	            //Year
	            #PieceID[23] := #is_ActualTime[1];
	            #PieceID[24] := #is_ActualTime[2];
	            #PieceID[25] := #is_ActualTime[3];
	            #PieceID[26] := #is_ActualTime[4];

	            //Month
	            #PieceID[27] := #is_ActualTime[6];
	            #PieceID[28] := #is_ActualTime[7];

	            //Day
	            #PieceID[29] := #is_ActualTime[9];
	            #PieceID[30] := #is_ActualTime[10];

	            //Constant
	            #PieceID[31] := '_';

	            //Time
	            #PieceID[32] := #is_ActualTime[12];
	            #PieceID[33] := #is_ActualTime[13];
	            #PieceID[34] := #is_ActualTime[14];
	            #PieceID[35] := #is_ActualTime[15];

	            //Constant
	            #PieceID[36] := '_';

	            //GIN
	            #ts_String := DELETE(IN := DINT_TO_STRING(#ii_GIN), L := 1, P := 1);

	            IF (#ii_GIN > 0) AND (#ii_GIN <= 9) THEN
	                #PieceID[37] := '0';
	                #PieceID[38] := '0';
	                #PieceID[39] := '0';
	                #PieceID[40] := #ts_String[1];
	            ELSIF (#ii_GIN >= 10) AND (#ii_GIN <= 99) THEN
	                #PieceID[37] := '0';
	                #PieceID[38] := '0';
	                #PieceID[39] := #ts_String[1];
	                #PieceID[40] := #ts_String[2];
	            ELSIF (#ii_GIN >= 100) AND (#ii_GIN <= 999) THEN
	                #PieceID[37] := '0';
	                #PieceID[38] := #ts_String[1];
	                #PieceID[39] := #ts_String[2];
	                #PieceID[40] := #ts_String[3];
	            ELSIF (#ii_GIN >= 1000) AND (#ii_GIN <= 9999) THEN
	                #PieceID[37] := #ts_String[1];
	                #PieceID[38] := #ts_String[2];
	                #PieceID[39] := #ts_String[3];
	                #PieceID[40] := #ts_String[4];
	            END_IF;

	            //Save data in DB GIN
	            "DB_GIN".GIN[#ii_GIN].DHL.PieceID := #PieceID;
	            "DB_GIN".GIN[#ii_GIN].DHL.VID := '000000000000000';

	            IF "DB_GIN".GIN[#ii_GIN].DHL.ObjectID = '' THEN
	                "DB_GIN".GIN[#ii_GIN].DHL.ObjectID := '0000000000';
	            END_IF;

	            //Generate a message to MFC
	            #FB_MFC_Sort_COY_ReceiveResult_Instance(is_VID := "DB_GIN".GIN[#ii_GIN].DHL.VID,
	                                                    is_PieceID := "DB_GIN".GIN[#ii_GIN].DHL.PieceID,
	                                                    is_Group := "DB_GIN".GIN[#ii_GIN].DHL.Xray.Group,
	                                                    is_Level := "DB_GIN".GIN[#ii_GIN].DHL.Xray.Level,
	                                                    is_Result := "DB_GIN".GIN[#ii_GIN].DHL.Xray.Result,
	                                                    ii_SourceNode := #ii_SourceNode,
	                                                    ii_DestinationNode := #ii_DestinationNode,
	                                                    iq_UDT_FifoHeader := #iq_UDT_FifoHeader,
	                                                    iqa_FifoData := #iqa_FifoData,
	                                                    iqi_MessageSequenceNumber := #iqi_MessageSequenceNumber);

	        END_IF;

	    END_IF;

	END_REGION

	REGION Parcel lost

	    //Check if parcel is lost in the tracking
	    //If there is, generate a message to MFC

	    IF #ii_GIN > 0 THEN

	        IF "DB_GIN".GIN[#ii_GIN].General.Lost THEN

	            //FORTNA internal exception results: L = Parcel lost
	            "DB_GIN".GIN[#ii_GIN].DHL.Xray.Result := 'L';

	            #FB_MFC_Sort_COY_ReceiveResult_Instance(is_VID := "DB_GIN".GIN[#ii_GIN].DHL.VID,
	                                                    is_PieceID := "DB_GIN".GIN[#ii_GIN].DHL.PieceID,
	                                                    is_Group := "DB_GIN".GIN[#ii_GIN].DHL.Xray.Group,
	                                                    is_Level := "DB_GIN".GIN[#ii_GIN].DHL.Xray.Level,
	                                                    is_Result := "DB_GIN".GIN[#ii_GIN].DHL.Xray.Result,
	                                                    ii_SourceNode := #ii_SourceNode,
	                                                    ii_DestinationNode := #ii_DestinationNode,
	                                                    iq_UDT_FifoHeader := #iq_UDT_FifoHeader,
	                                                    iqa_FifoData := #iqa_FifoData,
	                                                    iqi_MessageSequenceNumber := #iqi_MessageSequenceNumber);

	            //Save info in DB_GIN
	            "DB_GIN".GIN[#ii_GIN].DHL.MFCMessage.Sent.XrayResult := True;

	        END_IF;

	    END_IF;

	END_REGION

END_FUNCTION_BLOCK

FUNCTION_BLOCK "FB_MergeGINandObjectID"
{ S7_Optimized_Access := 'TRUE' }
VERSION : 0.1
// ATTRIBUTES
// AUTO_NUMBER = True
// BLOCK_NUMBER = 240
// END_ATTRIBUTES
   VAR_INPUT
      is_Configuration { ExternalAccessible := 'False'; ExternalVisible := 'False'; ExternalWritable := 'False'} : Struct   // Configuration
         SearchWindowStart { ExternalAccessible := 'False'; ExternalVisible := 'False'; ExternalWritable := 'False'} : Int;   // Start of the search window in conveyor tracking
         SearchWindowEnd { ExternalAccessible := 'False'; ExternalVisible := 'False'; ExternalWritable := 'False'} : Int;   // End of the search window in conveyor tracking
      END_STRUCT;
      iid_ReceivedObjectID { ExternalAccessible := 'False'; ExternalVisible := 'False'; ExternalWritable := 'False'} : DInt;   // Received ObjectID form sorter
      ia_ConveyorTracking { ExternalAccessible := 'False'; ExternalVisible := 'False'; ExternalWritable := 'False'} : Array[0..2501] of Int;   // ConveyorTracking
      ii_XrayLocation { ExternalAccessible := 'False'; ExternalVisible := 'False'; ExternalWritable := 'False'} : Int;   // X-ray location
      ii_SourceNode { ExternalAccessible := 'False'; ExternalVisible := 'False'; ExternalWritable := 'False'} : Int;   // ID Source Node
      ii_DestinationNode { ExternalAccessible := 'False'; ExternalVisible := 'False'; ExternalWritable := 'False'} : Int;   // ID Destination Node
   END_VAR

   VAR_IN_OUT
      iq_UDT_FifoHeader : "UDT_FifoHeader";   // FIFO header
      iqa_FifoData : Array[*] of "UDT_MessageV2";   // FIFO data buffer
      iqi_MessageSequenceNumber { ExternalAccessible := 'False'; ExternalVisible := 'False'; ExternalWritable := 'False'} : Int;   // Message number
   END_VAR

   VAR
      sid_ObjectID { ExternalAccessible := 'False'; ExternalVisible := 'False'; ExternalWritable := 'False'} : DInt;   // Saved Object ID
      sx_NewObjectID { ExternalAccessible := 'False'; ExternalVisible := 'False'; ExternalWritable := 'False'} : Bool;
      FB_MFC_Sort_COY_RegInfo_Instance { ExternalAccessible := 'False'; ExternalVisible := 'False'; ExternalWritable := 'False'; S7_SetPoint := 'False'} : "FB_MFC_Sort_COY_RegInfo";
   END_VAR

   VAR_TEMP
      ti_Loop : Int;
   END_VAR


BEGIN
	(*
	----------------------------------------------------------------------------------------
	|                                                                                      |
	|  Copyright  2023             FORTNA Europe BV                                        |
	|  All Rights Reserved         Netherlands                                             |
	|                                                                                      |
	----------------------------------------------------------------------------------------
	Version history:
	Date        | Version   | Author       | Remark
	----------------------------------------------------------------------------------------
	05/10/2023  | 1.0       | S. Nikodem   | Release TIA 17 | DHL Munich 2023
	13/03/2024  | 1.1       | S. Nieswiec  | Added to new Baseline
	*)

	REGION Save ObjectID

	    IF #iid_ReceivedObjectID <> #sid_ObjectID THEN

	        //New data
	        #sx_NewObjectID := True;

	        //Copy data to memory
	        #sid_ObjectID := #iid_ReceivedObjectID;

	    END_IF;

	END_REGION

	REGION Merge data

	    IF #sx_NewObjectID THEN

	        FOR #ti_Loop := #is_Configuration.SearchWindowStart TO #is_Configuration.SearchWindowEnd DO

	            IF #ia_ConveyorTracking[#ti_Loop] <> 0
	                AND ("DB_GIN".GIN[#ia_ConveyorTracking[#ti_Loop]].DHL.ObjectID = '')
	            THEN

	                //Combine data, save Object ID in DB GIN
	                "DB_GIN".GIN[#ia_ConveyorTracking[#ti_Loop]].DHL.ObjectID := DELETE(IN := DINT_TO_STRING(#sid_ObjectID), L := 1, P := 1);

	                //Data combined
	                #sx_NewObjectID := FALSE;

	                //Send a message to the MFC requesting information on the parcel
	                #FB_MFC_Sort_COY_RegInfo_Instance(is_ObjectID := "DB_GIN".GIN[#ia_ConveyorTracking[#ti_Loop]].DHL.ObjectID,
	                                                  ii_XrayLocation := #ii_XrayLocation,
	                                                  ii_SourceNode := #ii_SourceNode,
	                                                  ii_DestinationNode := #ii_DestinationNode,
	                                                  iq_UDT_FifoHeader := #iq_UDT_FifoHeader,
	                                                  iqa_FifoData := #iqa_FifoData,
	                                                  iqi_MessageSequenceNumber := #iqi_MessageSequenceNumber);

	                //Save information in DB GIN
	                "DB_GIN".GIN[#ia_ConveyorTracking[#ti_Loop]].DHL.MFCMessage.Sent.ParcelRegInfo := True;

	                //Exit loop
	                EXIT;

	            END_IF;

	        END_FOR;

	    END_IF;

	END_REGION
END_FUNCTION_BLOCK

FUNCTION_BLOCK "FB_SpecialHandlingArea"
TITLE = PLC0020 - DHL Munich
{ S7_Optimized_Access := 'TRUE' }
AUTHOR : 'R. Golonka'
VERSION : 0.1
// ATTRIBUTES
// AUTO_NUMBER = True
// BLOCK_NUMBER = 103
// END_ATTRIBUTES
//Block for special handling area
   VAR_INPUT
      i_UDT_ConveyorHandshakeUp { ExternalAccessible := 'False'; ExternalVisible := 'False'; ExternalWritable := 'False'} : "UDT_ConveyorHandshake";
      iudi_DelayTransferTime { ExternalAccessible := 'False'; ExternalVisible := 'False'; ExternalWritable := 'False'} : UDInt;   // Additional transfer time
      ix_KneeButton { ExternalAccessible := 'False'; ExternalVisible := 'False'; ExternalWritable := 'False'} : Bool;   // Input knee button conveyor 3
      ix_MannedButton { ExternalAccessible := 'False'; ExternalVisible := 'False'; ExternalWritable := 'False'} : Bool;   // Check in button to inform system about manned system
      ix_PEC_DownstreamEoS { ExternalAccessible := 'False'; ExternalVisible := 'False'; ExternalWritable := 'False'} : Bool;   // Downstream sensor end of section signal
      ix_PEC_EoS { ExternalAccessible := 'False'; ExternalVisible := 'False'; ExternalWritable := 'False'} : Bool;   // Sensor end of section signal
      ix_PEC_UpsteamEoS { ExternalAccessible := 'False'; ExternalVisible := 'False'; ExternalWritable := 'False'} : Bool;   // Upstream sensor end of section signal
      ix_LastStation { ExternalAccessible := 'False'; ExternalVisible := 'False'; ExternalWritable := 'False'} : Bool;   // Last station
   END_VAR

   VAR_OUTPUT
      q_UDT_HMIStatus { ExternalAccessible := 'False'; ExternalVisible := 'False'; ExternalWritable := 'False'} : "UDT_SHAStatus";   // SHA status
      qx_SygnalingLamp { ExternalAccessible := 'False'; ExternalVisible := 'False'; ExternalWritable := 'False'} : Bool;   // White lamp demmand
      qx_PushButtonLamp { ExternalAccessible := 'False'; ExternalVisible := 'False'; ExternalWritable := 'False'} : Bool;   // Push button lamp
      qx_ExternalDieback_1 { ExternalAccessible := 'False'; ExternalVisible := 'False'; ExternalWritable := 'False'} : Bool;   // External die back signal output
      qx_ExternalDieback_2 { ExternalAccessible := 'False'; ExternalVisible := 'False'; ExternalWritable := 'False'} : Bool;   // External die back signal output
      qx_ExternalDieback_3 { ExternalAccessible := 'False'; ExternalVisible := 'False'; ExternalWritable := 'False'} : Bool;   // External die back signal output
      qx_ExternalDiebackUp { ExternalAccessible := 'False'; ExternalVisible := 'False'; ExternalWritable := 'False'} : Bool;   // External die back signal output
   END_VAR

   VAR_IN_OUT
      iq_UDT_SHAInterfaceUp : "UDT_SHA_StationInterface";   // SHA interface
      iq_UDT_SHAInterface : "UDT_SHA_StationInterface";   // SHA interface
      iq_UDT_DownstreamConveyorHandshake : "UDT_ConveyorHandshake";   // Conveyor interface
      iq_UDT_ConveyorHandshake : "UDT_ConveyorHandshake";   // Conveyor interface
      iq_UDT_UpstreamConveyorHandshake : "UDT_ConveyorHandshake";   // Conveyor interface
   END_VAR

   VAR
      FB_TimerOnOffDelay_TransferInprogres { ExternalAccessible := 'False'; ExternalVisible := 'False'; ExternalWritable := 'False'; S7_SetPoint := 'False'} : "FB_TimerOnOffDelay";   // Additional timer time
      s_UDT_SHAInterface { ExternalAccessible := 'False'; ExternalVisible := 'False'; ExternalWritable := 'False'; S7_SetPoint := 'False'} : "UDT_SHA_StationInterface";   // Special handling area inteface
      s_UDT_HMIStatus { ExternalAccessible := 'False'; ExternalVisible := 'False'; ExternalWritable := 'False'; S7_SetPoint := 'False'} : "UDT_SHAStatus";   // SHA status
      R_TRIG_KneeButton {InstructionName := 'R_TRIG'; LibVersion := '1.0'; ExternalAccessible := 'False'; ExternalVisible := 'False'; ExternalWritable := 'False'; S7_SetPoint := 'False'} : R_TRIG;   // Rising edge knee button signal
      R_TRIG_MannedButton {InstructionName := 'R_TRIG'; LibVersion := '1.0'; ExternalAccessible := 'False'; ExternalVisible := 'False'; ExternalWritable := 'False'; S7_SetPoint := 'False'} : R_TRIG;   // Rising edge manned button signal
      R_TRIG_TIPUp {InstructionName := 'R_TRIG'; LibVersion := '1.0'; ExternalAccessible := 'False'; ExternalVisible := 'False'; ExternalWritable := 'False'; S7_SetPoint := 'False'} : R_TRIG;
      R_TRIG_TIPDown {InstructionName := 'R_TRIG'; LibVersion := '1.0'; ExternalAccessible := 'False'; ExternalVisible := 'False'; ExternalWritable := 'False'; S7_SetPoint := 'False'} : R_TRIG;
      R_TRIG_TIP {InstructionName := 'R_TRIG'; LibVersion := '1.0'; ExternalAccessible := 'False'; ExternalVisible := 'False'; ExternalWritable := 'False'; S7_SetPoint := 'False'} : R_TRIG;
      "#R_TRIG_RTSUp" {InstructionName := 'R_TRIG'; LibVersion := '1.0'; ExternalAccessible := 'False'; ExternalVisible := 'False'; ExternalWritable := 'False'; S7_SetPoint := 'False'} : R_TRIG;
      sx_SygnalingLamp { ExternalAccessible := 'False'; ExternalVisible := 'False'; ExternalWritable := 'False'} : Bool;   // White lamp demmand
      sx_PushButtonLamp { ExternalAccessible := 'False'; ExternalVisible := 'False'; ExternalWritable := 'False'} : Bool;   // Push button lamp
      sx_ExternalDieback_1 { ExternalAccessible := 'False'; ExternalVisible := 'False'; ExternalWritable := 'False'} : Bool;   // External dieback signal
      sx_ExternalDieback_2 { ExternalAccessible := 'False'; ExternalVisible := 'False'; ExternalWritable := 'False'} : Bool;   // External dieback signal
      sx_ExternalDieback_3 { ExternalAccessible := 'False'; ExternalVisible := 'False'; ExternalWritable := 'False'} : Bool;   // External dieback signal
      sx_ProductIsLocked { ExternalAccessible := 'False'; ExternalVisible := 'False'; ExternalWritable := 'False'} : Bool;   // Product is locked to the station
      sx_StationManned { ExternalAccessible := 'False'; ExternalVisible := 'False'; ExternalWritable := 'False'} : Bool;   // Station is occupied
      sx_DownstreamConveyorOccupied { ExternalAccessible := 'False'; ExternalVisible := 'False'; ExternalWritable := 'False'} : Bool;   // Downstream conveyor is occupied
      sx_MiddleConveyorOccupied { ExternalAccessible := 'False'; ExternalVisible := 'False'; ExternalWritable := 'False'} : Bool;   // Middle conveyor is occupied
      sx_UpstreamConveyorOccupied { ExternalAccessible := 'False'; ExternalVisible := 'False'; ExternalWritable := 'False'} : Bool;   // Upsteram conveyor is occupied
      si_NumberOfParcel { ExternalAccessible := 'False'; ExternalVisible := 'False'; ExternalWritable := 'False'} : Int;   // Number of parcel
      sx_ParcelTransfer { ExternalAccessible := 'False'; ExternalVisible := 'False'; ExternalWritable := 'False'} : Bool;   // Transfer in one section is in progress
      sx_ExternalDiebackUp { ExternalAccessible := 'False'; ExternalVisible := 'False'; ExternalWritable := 'False'} : Bool;   // Die back to previous station
   END_VAR


BEGIN
	(*
	----------------------------------------------------------------------------------------
	|                                                                                      |
	|  Copyright  2023             FORTNA Europe BV                                        |
	|  All Rights Reserved         Netherlands                                             |
	|                                                                                      |
	----------------------------------------------------------------------------------------
	Version history:
	Date        | Version   | Author       | Remark
	----------------------------------------------------------------------------------------
	06/10/2023  | 1.0       | R. Golonka   | Release TIA 17 | DHL Munich 2023
	13/03/2024  | 1.1       | S. Nieswiec  | Added to new baseline, block needs uptade after munich is finished
	*)

	REGION 1.0 - Inicialization
	    // Inicialization

	    #R_TRIG_KneeButton(CLK := #ix_KneeButton);
	    #R_TRIG_MannedButton(CLK := #ix_MannedButton);
	    #R_TRIG_TIPUp(CLK := #iq_UDT_UpstreamConveyorHandshake.TIP);
	    #R_TRIG_TIPDown(CLK := #iq_UDT_DownstreamConveyorHandshake.TIP);
	    #R_TRIG_TIP(CLK := #iq_UDT_ConveyorHandshake.TIP);
	    #"#R_TRIG_RTSUp"(CLK := #iq_UDT_ConveyorHandshake.RTS);

	END_REGION

	REGION 2.0 - Station manned

	    // Station in occupied (operator is working)
	    IF #R_TRIG_MannedButton.Q AND #iq_UDT_SHAInterfaceUp.Manned THEN

	        #sx_StationManned := NOT #sx_StationManned;
	        #sx_PushButtonLamp := NOT #sx_PushButtonLamp;

	    ELSIF (#iq_UDT_SHAInterfaceUp.Manned = false) THEN

	        #sx_StationManned := FALSE;
	        #sx_PushButtonLamp := FALSE;

	    ELSIF #ix_LastStation THEN

	        #sx_StationManned := #ix_LastStation;
	        #sx_PushButtonLamp := FALSE;

	    END_IF;

	END_REGION

	REGION 3.0 - Product locked and unlocked

	    // Product is locked in to the station
	    IF #R_TRIG_KneeButton.Q AND #sx_StationManned AND NOT #ix_PEC_DownstreamEoS THEN

	        #sx_ProductIsLocked := NOT #sx_ProductIsLocked;
	        #sx_SygnalingLamp := NOT #sx_SygnalingLamp;
	    ELSIF #R_TRIG_KneeButton.Q AND #sx_StationManned THEN
	        #sx_ProductIsLocked := false;
	        #sx_SygnalingLamp := false;
	    END_IF;

	END_REGION

	REGION 4.0 - Parcel in station

	    // Downstream station is occupied
	    #sx_DownstreamConveyorOccupied := NOT #ix_PEC_DownstreamEoS;
	    #sx_MiddleConveyorOccupied := NOT #ix_PEC_EoS;
	    #sx_UpstreamConveyorOccupied := NOT #ix_PEC_UpsteamEoS;

	    IF (#sx_DownstreamConveyorOccupied OR #sx_ProductIsLocked) THEN
	        #si_NumberOfParcel := 1;
	    END_IF;

	    IF (#sx_MiddleConveyorOccupied AND (#sx_DownstreamConveyorOccupied OR #sx_ProductIsLocked)) THEN
	        #si_NumberOfParcel := 2;
	    END_IF;

	    IF (#sx_UpstreamConveyorOccupied AND #sx_MiddleConveyorOccupied AND (#sx_DownstreamConveyorOccupied OR #sx_ProductIsLocked)) THEN
	        #si_NumberOfParcel := 3;
	    END_IF;

	    IF NOT #sx_UpstreamConveyorOccupied AND NOT #sx_MiddleConveyorOccupied AND NOT #sx_DownstreamConveyorOccupied THEN
	        #si_NumberOfParcel := 0;
	    END_IF;

	END_REGION

	REGION 5.0 - External dieback

	    IF #sx_StationManned
	        AND (#si_NumberOfParcel >= 3)
	        AND (#iq_UDT_SHAInterfaceUp.NumberOfParcel >= #si_NumberOfParcel)
	        AND #s_UDT_SHAInterface.Conveyor[2].Occupied
	        AND #s_UDT_SHAInterface.Conveyor[1].Occupied

	        OR #iq_UDT_SHAInterfaceUp.Conveyor[1].Locked
	        OR #sx_ProductIsLocked
	    THEN
	        #sx_ExternalDieback_1 := TRUE;
	    ELSE
	        #sx_ExternalDieback_1 := FALSE;
	    END_IF;

	    IF #sx_StationManned
	        AND (#si_NumberOfParcel >= 2)
	        AND (#iq_UDT_SHAInterfaceUp.NumberOfParcel >= #si_NumberOfParcel)
	        AND #s_UDT_SHAInterface.Conveyor[1].Occupied

	        OR #iq_UDT_SHAInterfaceUp.Conveyor[1].Locked
	        OR #sx_ProductIsLocked
	    THEN
	        #sx_ExternalDieback_2 := TRUE;
	    ELSE
	        #sx_ExternalDieback_2 := FALSE;
	    END_IF;

	    IF #sx_StationManned
	        AND (#si_NumberOfParcel >= 1)
	        AND (#iq_UDT_SHAInterfaceUp.NumberOfParcel >= #si_NumberOfParcel)
	        AND NOT #ix_PEC_DownstreamEoS
	        AND #iq_UDT_SHAInterfaceUp.Conveyor[1].Occupied
	        //AND #iq_UDT_SHAInterfaceUp.NumberOfParcel <> 0
	        OR #iq_UDT_SHAInterfaceUp.Conveyor[1].Locked
	        OR #sx_ProductIsLocked
	    THEN
	        #sx_ExternalDieback_3 := TRUE;
	    ELSIF #sx_StationManned AND (NOT #ix_PEC_DownstreamEoS AND #ix_LastStation) THEN
	        #sx_ExternalDieback_3 := TRUE;
	    ELSE
	        #sx_ExternalDieback_3 := FALSE;
	    END_IF;

	END_REGION

	REGION 8.0 - Reset RTR

	    // Set RTR to run conveyor

	    IF NOT #sx_DownstreamConveyorOccupied AND #ix_KneeButton AND #sx_StationManned THEN
	        #iq_UDT_DownstreamConveyorHandshake.RTR := true;
	    END_IF;

	    IF NOT #sx_MiddleConveyorOccupied AND #ix_KneeButton AND #sx_StationManned THEN
	        #iq_UDT_ConveyorHandshake.RTR := true;
	    END_IF;

	    IF NOT #sx_UpstreamConveyorOccupied AND #ix_KneeButton AND #sx_StationManned THEN
	        #iq_UDT_UpstreamConveyorHandshake.RTR := true;
	    END_IF;

	END_REGION

	REGION 7.0 - Hold for previous station when station is in transfer

	    #sx_ParcelTransfer := (#R_TRIG_KneeButton.Q)
	    OR (#R_TRIG_TIPDown.Q)
	    OR (#R_TRIG_TIP.Q)
	    OR (#R_TRIG_TIPUp.Q);

	    #FB_TimerOnOffDelay_TransferInprogres(iudi_OffDelayTime := #iudi_DelayTransferTime,
	                                          ix_SignalToDelay := #sx_ParcelTransfer,
	                                          ix_Enable := TRUE,
	                                          qx_DelayedSignal => #sx_ExternalDiebackUp);

	END_REGION

	REGION 8.0 - Update Interface

	    #s_UDT_SHAInterface.Manned := #sx_StationManned;
	    #s_UDT_SHAInterface.NumberOfParcel := #si_NumberOfParcel;
	    #s_UDT_SHAInterface.TransferInProgres := #sx_ParcelTransfer;
	    #s_UDT_SHAInterface.Conveyor[1].Empty := NOT #sx_DownstreamConveyorOccupied;
	    #s_UDT_SHAInterface.Conveyor[1].Locked := #sx_ProductIsLocked;
	    #s_UDT_SHAInterface.Conveyor[1].Occupied := #sx_DownstreamConveyorOccupied;
	    #s_UDT_SHAInterface.Conveyor[2].Empty := NOT #sx_MiddleConveyorOccupied;
	    #s_UDT_SHAInterface.Conveyor[2].Locked := FALSE;
	    #s_UDT_SHAInterface.Conveyor[2].Occupied := #sx_MiddleConveyorOccupied;
	    #s_UDT_SHAInterface.Conveyor[3].Empty := NOT #sx_UpstreamConveyorOccupied;
	    #s_UDT_SHAInterface.Conveyor[3].Locked := FALSE;
	    #s_UDT_SHAInterface.Conveyor[3].Occupied := #sx_UpstreamConveyorOccupied;

	END_REGION

	REGION 9.0 - Status

	    // Status half full
	    #s_UDT_HMIStatus.Specific.HalfFull := #sx_StationManned AND (#s_UDT_SHAInterface.NumberOfParcel >= 3);
	    // Status full
	    #s_UDT_HMIStatus.Specific.Full := #sx_StationManned AND (#iq_UDT_SHAInterfaceUp.NumberOfParcel >= 3) AND (#s_UDT_SHAInterface.NumberOfParcel >= 3) AND #i_UDT_ConveyorHandshakeUp.RTS;

	    // HMI status initialization
	    #s_UDT_HMIStatus.Status := 0;

	    // Copy HMI status to output
	    #q_UDT_HMIStatus := #s_UDT_HMIStatus;

	END_REGION

	REGION 10.0 - Output

	    // Output write
	    #qx_ExternalDieback_1 := #sx_ExternalDieback_1;
	    #qx_ExternalDieback_2 := #sx_ExternalDieback_2;
	    #qx_ExternalDieback_3 := #sx_ExternalDieback_3;
	    #qx_ExternalDiebackUp := #sx_ExternalDiebackUp AND #i_UDT_ConveyorHandshakeUp.RTS;
	    #qx_SygnalingLamp := #sx_SygnalingLamp;
	    #qx_PushButtonLamp := #sx_PushButtonLamp;
	    #iq_UDT_SHAInterface := #s_UDT_SHAInterface;

	END_REGION
END_FUNCTION_BLOCK

FUNCTION_BLOCK "FB_SNCY_InfeedControlPanel"
{ S7_Optimized_Access := 'TRUE' }
VERSION : 0.1
// ATTRIBUTES
// AUTO_NUMBER = True
// BLOCK_NUMBER = 102
// END_ATTRIBUTES
   VAR_INPUT
      ix_InfeedButton { ExternalAccessible := 'False'; ExternalVisible := 'False'; ExternalWritable := 'False'} : Bool;   // Signal from infeed push button
      ix_OutfeedButton { ExternalAccessible := 'False'; ExternalVisible := 'False'; ExternalWritable := 'False'} : Bool;   // Signal from outfeed push button
      i_UDT_ExitConveyorStatus { ExternalAccessible := 'False'; ExternalVisible := 'False'; ExternalWritable := 'False'} : "UDT_CommonStatus";   // Common status from outfeed exit conveyor
      ix_InfeedModeActive { ExternalAccessible := 'False'; ExternalVisible := 'False'; ExternalWritable := 'False'} : Bool;   // True - when infeed mode is active
      ix_OutfeedModeActive { ExternalAccessible := 'False'; ExternalVisible := 'False'; ExternalWritable := 'False'} : Bool;   // True - when outfeed mode is active
   END_VAR

   VAR_OUTPUT
      qx_InfeedLamp { ExternalAccessible := 'False'; ExternalVisible := 'False'; ExternalWritable := 'False'} : Bool;   // Lamp for Infeed status
      qx_OutfeedLamp { ExternalAccessible := 'False'; ExternalVisible := 'False'; ExternalWritable := 'False'} : Bool;   // Lamp for Outfeed status
      qx_ConveyorHold { ExternalAccessible := 'False'; ExternalVisible := 'False'; ExternalWritable := 'False'} : Bool;   // Conveyor hold command for associated conveyor
   END_VAR

   VAR
      R_TRIG_ToogleInfeedButton {InstructionName := 'R_TRIG'; LibVersion := '1.0'; ExternalAccessible := 'False'; ExternalVisible := 'False'; ExternalWritable := 'False'; S7_SetPoint := 'False'} : R_TRIG;   // Rising edge trigger infeed button
      R_TRIG_ToogleOutfeedButton {InstructionName := 'R_TRIG'; LibVersion := '1.0'; ExternalAccessible := 'False'; ExternalVisible := 'False'; ExternalWritable := 'False'; S7_SetPoint := 'False'} : R_TRIG;   // Rising edge trigger outfeed button
      R_TRIG_Modeline {InstructionName := 'R_TRIG'; LibVersion := '1.0'; ExternalAccessible := 'False'; ExternalVisible := 'False'; ExternalWritable := 'False'; S7_SetPoint := 'False'} : R_TRIG;   // Rising edge trigger mode line
      sx_SectionHold { ExternalAccessible := 'False'; ExternalVisible := 'False'; ExternalWritable := 'False'} : Bool;
   END_VAR


BEGIN
	(*
	----------------------------------------------------------------------------------------
	|                                                                                      |
	|  Copyright  2023             Fortna Europe BV                                        |
	|  All Rights Reserved         Netherlands                                             |
	|                                                                                      |
	|                                                                                      |
	----------------------------------------------------------------------------------------

	Version history:
	Date        | Version   | Author       | Remark
	----------------------------------------------------------------------------------------
	18/10/2023  | 1.0       | S. Nikodem   | Release TIA 17 | DHL Munich 2023
	13/03/2024  | 1.1       | S. Nieswiec  | Added to new baseline, block needs uptade after munich is finished
	*)

	REGION Buttons

	    //Infeed
	    IF #ix_InfeedModeActive THEN

	        #R_TRIG_ToogleInfeedButton(CLK := (#ix_InfeedButton));

	        IF #R_TRIG_ToogleInfeedButton.Q THEN

	            #sx_SectionHold := NOT #sx_SectionHold;

	        END_IF;

	    END_IF;

	    //Outfeed
	    IF #ix_OutfeedModeActive THEN

	        #R_TRIG_ToogleOutfeedButton(CLK := (#ix_OutfeedButton));

	        IF #R_TRIG_ToogleOutfeedButton.Q THEN

	            #sx_SectionHold := NOT #sx_SectionHold;

	        END_IF;

	    END_IF;

	END_REGION

	REGION Lamps

	    //Infeed
	    IF #ix_InfeedModeActive THEN

	        IF #sx_SectionHold THEN
	            #qx_InfeedLamp := "DB_Memory".Clock_1Hz;
	        ELSE
	            #qx_InfeedLamp := TRUE;
	        END_IF;

	    ELSE
	        #qx_InfeedLamp := False;
	    END_IF;

	    //Outfeed
	    IF #ix_OutfeedModeActive THEN

	        IF #sx_SectionHold THEN
	            #qx_OutfeedLamp := "DB_Memory".Clock_1Hz;
	        ELSE
	            #qx_OutfeedLamp := TRUE;
	        END_IF;

	    ELSE
	        #qx_OutfeedLamp := False;
	    END_IF;

	END_REGION

	REGION Conveyor hold command

	    #qx_ConveyorHold := #sx_SectionHold;

	END_REGION

	REGION Reset

	    //Reset when mode line is changed
	    #R_TRIG_Modeline(CLK := #ix_InfeedModeActive OR #ix_OutfeedModeActive);

	    IF #R_TRIG_Modeline.Q THEN
	        // Statement section IF
	        ;
	    END_IF;


	END_REGION



END_FUNCTION_BLOCK

FUNCTION_BLOCK "FB_SNCY_ArmDiverter"
{ S7_Optimized_Access := 'TRUE' }
VERSION : 0.1
// ATTRIBUTES
// AUTO_NUMBER = True
// BLOCK_NUMBER = 241
// END_ATTRIBUTES
   VAR_INPUT
      i_UDT_DiverterArmConfig { ExternalAccessible := 'False'; ExternalVisible := 'False'; ExternalWritable := 'False'} : "UDT_ArmDiverterConfiguration";   // Diverter arm configuration
      ix_SafetyOk { ExternalAccessible := 'False'; ExternalVisible := 'False'; ExternalWritable := 'False'} : Bool;   // TRUE when safety is ok
      ix_24vOk { ExternalAccessible := 'False'; ExternalVisible := 'False'; ExternalWritable := 'False'} : Bool;   // TRUE when 24VDC is healthy
      ix_400vOk { ExternalAccessible := 'False'; ExternalVisible := 'False'; ExternalWritable := 'False'} : Bool;   // TRUE when 400VAC is healthy
      ix_HardwareOk { ExternalAccessible := 'False'; ExternalVisible := 'False'; ExternalWritable := 'False'} : Bool;   // TRUE when  hardware is Ok
      ix_PRX_Home { ExternalAccessible := 'False'; ExternalVisible := 'False'; ExternalWritable := 'False'} : Bool;   // Proxy sensor home position
      ix_PRX_Divert { ExternalAccessible := 'False'; ExternalVisible := 'False'; ExternalWritable := 'False'} : Bool;   // Proxy sensor divert position
      ix_LS_Home { ExternalAccessible := 'False'; ExternalVisible := 'False'; ExternalWritable := 'False'} : Bool;   // Limit switch home position
      ix_LS_Divert { ExternalAccessible := 'False'; ExternalVisible := 'False'; ExternalWritable := 'False'} : Bool;   // Limit switch divert position
      ix_PRX_BRK_Home { ExternalAccessible := 'False'; ExternalVisible := 'False'; ExternalWritable := 'False'} : Bool;   // Brake sensor divert
      ix_PRX_BRK_Divert { ExternalAccessible := 'False'; ExternalVisible := 'False'; ExternalWritable := 'False'} : Bool;   // Brake sensor home
      ix_PEC_Exit { ExternalAccessible := 'False'; ExternalVisible := 'False'; ExternalWritable := 'False'} : Bool;   // TRUE when PEC Exit is not blocked
      ii_SourceNode { ExternalAccessible := 'False'; ExternalVisible := 'False'; ExternalWritable := 'False'} : Int := 0;   // Source Node
      ii_DestinationNode { ExternalAccessible := 'False'; ExternalVisible := 'False'; ExternalWritable := 'False'} : Int := 0;   // Destination Node
   END_VAR

   VAR_OUTPUT
      q_UDT_HMIStatus { ExternalAccessible := 'False'; ExternalVisible := 'False'; ExternalWritable := 'False'} : "UDT_ArmDiverterStatus";   // HMI status structure
      q_UDT_Status { ExternalAccessible := 'False'; ExternalVisible := 'False'; ExternalWritable := 'False'} : "UDT_CommonStatus";   // Common status structure
      qx_VerticalConveyorHold { ExternalAccessible := 'False'; ExternalVisible := 'False'; ExternalWritable := 'False'} : Bool;   // Command stop Vertical conveyor
      qx_AssociatedConveyorHold { ExternalAccessible := 'False'; ExternalVisible := 'False'; ExternalWritable := 'False'} : Bool;   // Command stop Associated conveyor
   END_VAR

   VAR_IN_OUT
      iq_UDT_EquipmentControl : "UDT_EquipmentControl";   // Equipment control structure
      iq_UDT_AssociatedConveyorInterface : "UDT_ConveyorInterface";   // Sorter main conveyor interface
      iq_UDT_VerticalConveyorInterface : "UDT_ConveyorInterface";   // Arm vertical conveyor interafce
      iq_UDT_ArmConveyorInterface : "UDT_ConveyorInterface";   // Arm conveyor interface
      iq_UDT_AssociatedConveyorHandshake : "UDT_ConveyorHandshake";   // Handshake structure
      iq_UDT_ExitConveyorHandshake : "UDT_ConveyorHandshake";   // Exit conveyor handshake structure
      iqa_AssociatedTrackingData : Array[*] of Int;   // Tracking data from sorter conveyor
      iqa_OutfeedsStatus : Array[*] of "UDT_OutfeedStatus";   // Structure with outfeeds status
      iq_UDT_ArmDiverterCommand : "UDT_ArmDiverterCommand";   // Arm Diverter command structure
      iq_UDT_FifoHeader_MFCMessage : "UDT_FifoHeader";   // MFC Message FIFO header
      iqs_FifoData_MFCMessage : Array[*] of "UDT_MessageV2";   // MFC Message FIFO data buffer
      iqdi_MessageSequenceNumber { ExternalAccessible := 'False'; ExternalVisible := 'False'; ExternalWritable := 'False'} : Int;   // MFC Message Message number
   END_VAR

   VAR
      FB_MFC_Sort_SortResult_HigherPriorityAvailable { ExternalAccessible := 'False'; ExternalVisible := 'False'; ExternalWritable := 'False'; S7_SetPoint := 'False'} : "FB_MFC_Sort_SortResult";   // Function to MFC message generation
      FB_MFC_Sort_SortResult { ExternalAccessible := 'False'; ExternalVisible := 'False'; ExternalWritable := 'False'; S7_SetPoint := 'False'} : "FB_MFC_Sort_SortResult";   // Function to MFC message generation
      FB_MFC_Sort_SortResult_Instance { ExternalAccessible := 'False'; ExternalVisible := 'False'; ExternalWritable := 'False'; S7_SetPoint := 'False'} : "FB_MFC_Sort_SortResult";   // Function to MFC message generation
      s_FB_PRX_HomeFiltered { ExternalAccessible := 'False'; ExternalVisible := 'False'; ExternalWritable := 'False'; S7_SetPoint := 'False'} : "FB_TimerOnOffDelay";   // Filtering proxy sensor home position signal
      s_FB_PRX_DivertFiltered { ExternalAccessible := 'False'; ExternalVisible := 'False'; ExternalWritable := 'False'; S7_SetPoint := 'False'} : "FB_TimerOnOffDelay";   // Filtering proxy sensor divert position signal
      s_FB_LS_HomeFiltered { ExternalAccessible := 'False'; ExternalVisible := 'False'; ExternalWritable := 'False'; S7_SetPoint := 'False'} : "FB_TimerOnOffDelay";   // Filtering limit switch home position signal
      s_FB_LS_DivertFiltered { ExternalAccessible := 'False'; ExternalVisible := 'False'; ExternalWritable := 'False'; S7_SetPoint := 'False'} : "FB_TimerOnOffDelay";   // Filtering limit switch divert position signal
      s_FB_BRK_PRX_HomeFiltered { ExternalAccessible := 'False'; ExternalVisible := 'False'; ExternalWritable := 'False'; S7_SetPoint := 'False'} : "FB_TimerOnOffDelay";   // Filtering proxy sensor home position signal
      s_FB_BRK_PRX_DivertFiltered { ExternalAccessible := 'False'; ExternalVisible := 'False'; ExternalWritable := 'False'; S7_SetPoint := 'False'} : "FB_TimerOnOffDelay";   // Filtering proxy sensor divert position signal
      s_FB_TimeoutError { ExternalAccessible := 'False'; ExternalVisible := 'False'; ExternalWritable := 'False'; S7_SetPoint := 'False'} : "FB_TimerOnOffDelay";   // Movement timeout error
      s_FB_Jog_Enable { ExternalAccessible := 'False'; ExternalVisible := 'False'; ExternalWritable := 'False'; S7_SetPoint := 'False'} : "FB_TimerOnOffDelay";   // Filtering lower jam photo eye signal
      s_FB_DivertTime { ExternalAccessible := 'False'; ExternalVisible := 'False'; ExternalWritable := 'False'; S7_SetPoint := 'False'} : "FB_TimerOnOffDelay";   // Divert time
      s_FB_InhibitTimeFilter { ExternalAccessible := 'False'; ExternalVisible := 'False'; ExternalWritable := 'False'; S7_SetPoint := 'False'} : "FB_TimerOnOffDelay";   // Filtering inhibit stop
      s_UDT_CommonStatus { ExternalAccessible := 'False'; ExternalVisible := 'False'; ExternalWritable := 'False'; S7_SetPoint := 'False'} : "UDT_CommonStatus";   // Common status structure
      s_UDT_CommonStatusOld { ExternalAccessible := 'False'; ExternalVisible := 'False'; ExternalWritable := 'False'; S7_SetPoint := 'False'} : "UDT_CommonStatus";   // Auxiliary status structure
      s_UDT_HMIStatus { ExternalAccessible := 'False'; ExternalVisible := 'False'; ExternalWritable := 'False'; S7_SetPoint := 'False'} : "UDT_ArmDiverterStatus";   // HMI status structure
      R_TRIG_ManualJogHome {InstructionName := 'R_TRIG'; LibVersion := '1.0'; ExternalAccessible := 'False'; ExternalVisible := 'False'; ExternalWritable := 'False'; S7_SetPoint := 'False'} : R_TRIG;   // Rising edge trigger manual jog mode command
      R_TRIG_ManualJogDivert {InstructionName := 'R_TRIG'; LibVersion := '1.0'; ExternalAccessible := 'False'; ExternalVisible := 'False'; ExternalWritable := 'False'; S7_SetPoint := 'False'} : R_TRIG;   // Rising edge trigger manual jog mode command
      R_TRIG_PRX_Home {InstructionName := 'R_TRIG'; LibVersion := '1.0'; ExternalAccessible := 'False'; ExternalVisible := 'False'; ExternalWritable := 'False'; S7_SetPoint := 'False'} : R_TRIG;   // Rising edge trigger
      R_TRIG_PRX_Divert {InstructionName := 'R_TRIG'; LibVersion := '1.0'; ExternalAccessible := 'False'; ExternalVisible := 'False'; ExternalWritable := 'False'; S7_SetPoint := 'False'} : R_TRIG;   // Rising edge trigger
      R_TRIG_LS_Home {InstructionName := 'R_TRIG'; LibVersion := '1.0'; ExternalAccessible := 'False'; ExternalVisible := 'False'; ExternalWritable := 'False'; S7_SetPoint := 'False'} : R_TRIG;   // Rising edge trigger
      R_TRIG_LS_Divert {InstructionName := 'R_TRIG'; LibVersion := '1.0'; ExternalAccessible := 'False'; ExternalVisible := 'False'; ExternalWritable := 'False'; S7_SetPoint := 'False'} : R_TRIG;   // Rising edge trigger
      F_TRIG_PRX_Home {InstructionName := 'F_TRIG'; LibVersion := '1.0'; ExternalAccessible := 'False'; ExternalVisible := 'False'; ExternalWritable := 'False'; S7_SetPoint := 'False'} : F_TRIG;   // Falling edge trigger
      F_TRIG_PRX_Divert {InstructionName := 'F_TRIG'; LibVersion := '1.0'; ExternalAccessible := 'False'; ExternalVisible := 'False'; ExternalWritable := 'False'; S7_SetPoint := 'False'} : F_TRIG;   // Falling edge trigger
      F_TRIG_LS_Home {InstructionName := 'F_TRIG'; LibVersion := '1.0'; ExternalAccessible := 'False'; ExternalVisible := 'False'; ExternalWritable := 'False'; S7_SetPoint := 'False'} : F_TRIG;   // Falling edge trigger
      F_TRIG_LS_Divert {InstructionName := 'F_TRIG'; LibVersion := '1.0'; ExternalAccessible := 'False'; ExternalVisible := 'False'; ExternalWritable := 'False'; S7_SetPoint := 'False'} : F_TRIG;   // Falling edge trigger
      F_TRIG_BRK_PRX_Home {InstructionName := 'F_TRIG'; LibVersion := '1.0'; ExternalAccessible := 'False'; ExternalVisible := 'False'; ExternalWritable := 'False'; S7_SetPoint := 'False'} : F_TRIG;   // Falling edge trigger
      R_TRIG_BRK_PRX_Home {InstructionName := 'R_TRIG'; LibVersion := '1.0'; ExternalAccessible := 'False'; ExternalVisible := 'False'; ExternalWritable := 'False'; S7_SetPoint := 'False'} : R_TRIG;   // Rising edge trigger
      F_TRIG_BRK_PRX_Divert {InstructionName := 'F_TRIG'; LibVersion := '1.0'; ExternalAccessible := 'False'; ExternalVisible := 'False'; ExternalWritable := 'False'; S7_SetPoint := 'False'} : F_TRIG;   // Falling edge trigger
      R_TRIG_BRK_PRX_Divert {InstructionName := 'R_TRIG'; LibVersion := '1.0'; ExternalAccessible := 'False'; ExternalVisible := 'False'; ExternalWritable := 'False'; S7_SetPoint := 'False'} : R_TRIG;   // Rising edge trigger
      R_TRIG_ExitSensor {InstructionName := 'R_TRIG'; LibVersion := '1.0'; ExternalAccessible := 'False'; ExternalVisible := 'False'; ExternalWritable := 'False'; S7_SetPoint := 'False'} : R_TRIG;   // Rising edge trigger of exit sensor
      F_TRIG_ArmConveyorLowSpeed {InstructionName := 'F_TRIG'; LibVersion := '1.0'; ExternalAccessible := 'False'; ExternalVisible := 'False'; ExternalWritable := 'False'; S7_SetPoint := 'False'} : F_TRIG;   // Falling edge trigger
      R_TRIG_ParcelLocation {InstructionName := 'R_TRIG'; LibVersion := '1.0'; ExternalAccessible := 'False'; ExternalVisible := 'False'; ExternalWritable := 'False'; S7_SetPoint := 'False'} : R_TRIG;   // Rising edge trigger
      ss_Counter { ExternalAccessible := 'False'; ExternalVisible := 'False'; ExternalWritable := 'False'} : Struct   // Counters for statistics
         ParcelDetected { ExternalAccessible := 'False'; ExternalVisible := 'False'; ExternalWritable := 'False'} : UDInt;   // New package was detected
         ParcelInWindow { ExternalAccessible := 'False'; ExternalVisible := 'False'; ExternalWritable := 'False'} : UDInt;   // Another parcel is within the range of arm movement. The parcel cannot be sorted.
         SortParcelCommand { ExternalAccessible := 'False'; ExternalVisible := 'False'; ExternalWritable := 'False'} : UDInt;
         SortResultMessage { ExternalAccessible := 'False'; ExternalVisible := 'False'; ExternalWritable := 'False'} : UDInt;
         LoopExit { ExternalAccessible := 'False'; ExternalVisible := 'False'; ExternalWritable := 'False'} : UDInt;
      END_STRUCT;
      ss_SortStrategy { ExternalAccessible := 'False'; ExternalVisible := 'False'; ExternalWritable := 'False'} : Struct   // Sort Strategy
         HigherPriorityAvailable { ExternalAccessible := 'False'; ExternalVisible := 'False'; ExternalWritable := 'False'} : Bool;
         ObjectID { ExternalAccessible := 'False'; ExternalVisible := 'False'; ExternalWritable := 'False'} : String[10];
      END_STRUCT;
      ss_SortedObjectID { ExternalAccessible := 'False'; ExternalVisible := 'False'; ExternalWritable := 'False'} : String[10];   // Stored value of the last Object ID
      si_GINSort { ExternalAccessible := 'False'; ExternalVisible := 'False'; ExternalWritable := 'False'} : Int := 1;   // GIN code
      si_OutfeedsNumber { ExternalAccessible := 'False'; ExternalVisible := 'False'; ExternalWritable := 'False'} : Int;   // Number of connected outfeeds
      si_SortParcelEndPositon { ExternalAccessible := 'False'; ExternalVisible := 'False'; ExternalWritable := 'False'} : Int;   // Sort parcel end positon
      si_DecisionPointGIN { ExternalAccessible := 'False'; ExternalVisible := 'False'; ExternalWritable := 'False'} : Int;   // Decision point GIN
      si_DecisionPointGINDistance { ExternalAccessible := 'False'; ExternalVisible := 'False'; ExternalWritable := 'False'} : Int;   // Decision point GIN distance
      si_LocationGIN { ExternalAccessible := 'False'; ExternalVisible := 'False'; ExternalWritable := 'False'} : Int;   // Location GIN
      sx_AutoArmDivert { ExternalAccessible := 'False'; ExternalVisible := 'False'; ExternalWritable := 'False'} : Bool;   // True - Command arm should turn to "Divert position", command generated in auto mode
      sx_AutoArmHome { ExternalAccessible := 'False'; ExternalVisible := 'False'; ExternalWritable := 'False'} : Bool;   // True - Command arm should turn to "Home position", command generated in auto mode
      sx_Ready { ExternalAccessible := 'False'; ExternalVisible := 'False'; ExternalWritable := 'False'} : Bool;   // Ready to operate in Automatic mode
      sx_NewParcel { ExternalAccessible := 'False'; ExternalVisible := 'False'; ExternalWritable := 'False'} : Bool;   // True - new parcel was detected
      sx_ConfigurationError { ExternalAccessible := 'False'; ExternalVisible := 'False'; ExternalWritable := 'False'} : Bool;   // True - the configuration error occured
      sx_ArmDiverterLowSpeed { ExternalAccessible := 'False'; ExternalVisible := 'False'; ExternalWritable := 'False'} : Bool;   // Arm diverter low speed
      sx_Disabled { ExternalAccessible := 'False'; ExternalVisible := 'False'; ExternalWritable := 'False'} : Bool;   // True - if the functionality is disabled
      sx_PiorityDestinationNOK { ExternalAccessible := 'False'; ExternalVisible := 'False'; ExternalWritable := 'False'} : Bool;   // True - when Previous destination unavailable
      sx_ActualArmPositionHome { ExternalAccessible := 'False'; ExternalVisible := 'False'; ExternalWritable := 'False'} : Bool;   // True - if the arm is set in the Home position
      sx_ActualArmPositionOnWay { ExternalAccessible := 'False'; ExternalVisible := 'False'; ExternalWritable := 'False'} : Bool;   // True - if the arm is set in the way on position
      sx_ActualArmPositionDivert { ExternalAccessible := 'False'; ExternalVisible := 'False'; ExternalWritable := 'False'} : Bool;   // True - if the arm is set in the Extended position
      sx_MoveToHomePosition { ExternalAccessible := 'False'; ExternalVisible := 'False'; ExternalWritable := 'False'} : Bool;   // Command in automatic mode - Move to home position
      sx_MoveToDivertPosition { ExternalAccessible := 'False'; ExternalVisible := 'False'; ExternalWritable := 'False'} : Bool;   // Command in automatic mode - Move to divert position
      sx_ManualToHomePosition { ExternalAccessible := 'False'; ExternalVisible := 'False'; ExternalWritable := 'False'} : Bool;   // Command in manual mode - Move to home position
      sx_ManualToDivertPosition { ExternalAccessible := 'False'; ExternalVisible := 'False'; ExternalWritable := 'False'} : Bool;   // Command in manual mode - Move to divert position
      sx_JogToHomePosition { ExternalAccessible := 'False'; ExternalVisible := 'False'; ExternalWritable := 'False'} : Bool;   // Command in jog mode - Move to home position
      sx_JogToDivertPosition { ExternalAccessible := 'False'; ExternalVisible := 'False'; ExternalWritable := 'False'} : Bool;   // Command in jog mode - Move to divert position
      sx_PRX_HomeFiltered { ExternalAccessible := 'False'; ExternalVisible := 'False'; ExternalWritable := 'False'} : Bool;   // Proxy sensor home position filtered
      sx_PRX_DivertFiltered { ExternalAccessible := 'False'; ExternalVisible := 'False'; ExternalWritable := 'False'} : Bool;   // Proxy sensor divert position filtered
      sx_LS_HomeFiltered { ExternalAccessible := 'False'; ExternalVisible := 'False'; ExternalWritable := 'False'} : Bool;   // Limit switch home position filtered
      sx_LS_DivertFiltered { ExternalAccessible := 'False'; ExternalVisible := 'False'; ExternalWritable := 'False'} : Bool;   // Limit switch divert position filtered
      sx_PRX_BRK_HomeFiltered { ExternalAccessible := 'False'; ExternalVisible := 'False'; ExternalWritable := 'False'} : Bool;   // Brake sensor home filtered
      sx_PRX_BRK_DivertFiltered { ExternalAccessible := 'False'; ExternalVisible := 'False'; ExternalWritable := 'False'} : Bool;   // Brake sensor divert filtered
      sx_SwitchEnable { ExternalAccessible := 'False'; ExternalVisible := 'False'; ExternalWritable := 'False'} : Bool;   // Switching conditions
      sx_ParcelSorted { ExternalAccessible := 'False'; ExternalVisible := 'False'; ExternalWritable := 'False'} : Bool;   // Parcel in area
      sx_LimitSwitchHomeReached { ExternalAccessible := 'False'; ExternalVisible := 'False'; ExternalWritable := 'False'} : Bool;   // Limit switch home reached
      sx_LimitSwitchDivertReached { ExternalAccessible := 'False'; ExternalVisible := 'False'; ExternalWritable := 'False'} : Bool;   // Limit switch divert reached
      sx_PositionHomeReached { ExternalAccessible := 'False'; ExternalVisible := 'False'; ExternalWritable := 'False'} : Bool;   // Position home reached
      sx_PositionDivertReached { ExternalAccessible := 'False'; ExternalVisible := 'False'; ExternalWritable := 'False'} : Bool;   // Position divert reached
      sx_ParcelInWindow { ExternalAccessible := 'False'; ExternalVisible := 'False'; ExternalWritable := 'False'} : Bool;   // Parcel in window
      sx_GenerationMessage { ExternalAccessible := 'False'; ExternalVisible := 'False'; ExternalWritable := 'False'} : Bool;   // Generation MFC message
   END_VAR

   VAR_TEMP
      ti_LoopOutfeeds : Int;   // Loop counter
      ti_LoopDestination : Int;   // Loop counter
      ti_LoopDestinationNearest : Int;   // Loop counter
      ti_LoopParcelFreeArea : Int;   // Loop counter
      ti_LoopParcel : Int;   // Loop counter
      ti_LoopResult : Int;   // Loop counter
      tx_MovementCommandActive : Bool;   // Movement command active
   END_VAR

   VAR CONSTANT
      ci_DestinationNumberMin : Int := 350;   // Minimum number of available destination
      ci_DestinationNumberMax : Int := 356;   // Maximum number of available destination
      ci_OutfeedNumberMax : Int := 6;   // Maximum number of Outfeeds
      cs_SortStrategyNearest : String := '2';   // Value of sort strategy nearest
      cs_SortStrategyHighestPriority : String := '1';   // Value of sort strategy highest priority
      cudi_InhibitTimeFilterTimeOFF : UDInt := 1500;   // Time to stop
   END_VAR


BEGIN
	(*
	----------------------------------------------------------------------------------------
	|                                                                                      |
	|  Copyright  2023             FORTNA Europe BV                                        |
	|  All Rights Reserved         Netherlands                                             |
	|                                                                                      |
	----------------------------------------------------------------------------------------
	Version history:
	Date        | Version   | Author       | Remark
	----------------------------------------------------------------------------------------
	06/06/2023  | 1.0       | S. Nikodem   | Release TIA 17 | DHL Munich 2023
	10/08/2023  | 1.1       | S. Nikodem   | Sort Strategy
	17/10/2023  | 1.2       | S. Nikodem   | Added brake sensors and local reset
	13/03/2024  | 1.3       | S. Nieswiec  | Added to new baseline, block needs uptade after munich is finished

	*)

	REGION 1 - Triggers / Filters

	    //Triggers
	    //Proxy sensor home position
	    //Rising edge trigger
	    #R_TRIG_PRX_Home(CLK := #sx_PRX_HomeFiltered);
	    //Falling edge trigger
	    #F_TRIG_PRX_Home(CLK := #sx_PRX_HomeFiltered);

	    //Proxy sensor divert position
	    //Rising edge trigger
	    #R_TRIG_PRX_Divert(CLK := #sx_PRX_DivertFiltered);
	    //Falling edge trigger
	    #F_TRIG_PRX_Divert(CLK := #sx_PRX_DivertFiltered);

	    //Limit switch home position
	    //Rising edge trigger
	    #R_TRIG_LS_Home(CLK := #sx_LS_HomeFiltered);
	    //Falling edge trigger
	    #F_TRIG_LS_Home(CLK := #sx_LS_HomeFiltered);

	    //Limit switch divert position
	    //Rising edge trigger
	    #R_TRIG_LS_Divert(CLK := #sx_LS_DivertFiltered);
	    //Falling edge trigger
	    #F_TRIG_LS_Divert(CLK := #sx_LS_DivertFiltered);

	    //Brake sensor home position
	    //Rising edge trigger
	    #R_TRIG_BRK_PRX_Home(CLK := #sx_PRX_BRK_HomeFiltered);
	    //Falling edge trigger
	    #F_TRIG_BRK_PRX_Home(CLK := #sx_PRX_BRK_HomeFiltered);

	    //Brake sensor divert position
	    //Rising edge trigger
	    #R_TRIG_BRK_PRX_Divert(CLK := #sx_PRX_BRK_DivertFiltered);
	    //Falling edge trigger
	    #F_TRIG_BRK_PRX_Divert(CLK := #sx_PRX_BRK_DivertFiltered);

	    //Exit sensor
	    #R_TRIG_ExitSensor(CLK := #ix_PEC_Exit);

	    //On/off Filters
	    //Proxy sensor home position
	    #s_FB_PRX_HomeFiltered(iudi_OnDelayTime := #i_UDT_DiverterArmConfig.Sensor.PRX_HomeTimeOnDelay,
	                           iudi_OffDelayTime := #i_UDT_DiverterArmConfig.Sensor.PRX_HomeTimeOffDelay,
	                           ix_SignalToDelay := #ix_PRX_Home,
	                           ix_Enable := TRUE,
	                           qx_DelayedSignal => #sx_PRX_HomeFiltered);

	    //Proxy sensor divert position
	    #s_FB_PRX_DivertFiltered(iudi_OnDelayTime := #i_UDT_DiverterArmConfig.Sensor.PRX_DivertTimeOnDelay,
	                             iudi_OffDelayTime := #i_UDT_DiverterArmConfig.Sensor.PRX_DivertTimeOffDelay,
	                             ix_SignalToDelay := #ix_PRX_Divert,
	                             ix_Enable := TRUE,
	                             qx_DelayedSignal => #sx_PRX_DivertFiltered);

	    //Limit switch home position
	    #s_FB_LS_HomeFiltered(iudi_OnDelayTime := #i_UDT_DiverterArmConfig.Sensor.LS_HomeTimeOnDelay,
	                          iudi_OffDelayTime := #i_UDT_DiverterArmConfig.Sensor.LS_HomeTimeOffDelay,
	                          ix_SignalToDelay := #ix_LS_Home,
	                          ix_Enable := TRUE,
	                          qx_DelayedSignal => #sx_LS_HomeFiltered);

	    //Limit switch divert position
	    #s_FB_LS_DivertFiltered(iudi_OnDelayTime := #i_UDT_DiverterArmConfig.Sensor.LS_DivertTimeOnDelay,
	                            iudi_OffDelayTime := #i_UDT_DiverterArmConfig.Sensor.LS_DivertTimeOffDelay,
	                            ix_SignalToDelay := #ix_LS_Divert,
	                            ix_Enable := TRUE,
	                            qx_DelayedSignal => #sx_LS_DivertFiltered);

	    //Brake sensor home
	    #s_FB_BRK_PRX_HomeFiltered(iudi_OnDelayTime := #i_UDT_DiverterArmConfig.Sensor.PRX_BRK_HomeTimeOnDelay,
	                               iudi_OffDelayTime := #i_UDT_DiverterArmConfig.Sensor.PRX_BRK_HomeTimeOffDelay,
	                               ix_SignalToDelay := #ix_PRX_BRK_Home,
	                               ix_Enable := TRUE,
	                               qx_DelayedSignal => #sx_PRX_BRK_HomeFiltered);

	    //Brake sensor divert
	    #s_FB_BRK_PRX_DivertFiltered(iudi_OnDelayTime := #i_UDT_DiverterArmConfig.Sensor.PRX_BRK_DivertTimeOnDelay,
	                                 iudi_OffDelayTime := #i_UDT_DiverterArmConfig.Sensor.PRX_BRK_DivertTimeOffDelay,
	                                 ix_SignalToDelay := #ix_PRX_BRK_Divert,
	                                 ix_Enable := TRUE,
	                                 qx_DelayedSignal => #sx_PRX_BRK_DivertFiltered);

	END_REGION

	REGION 2 - Configuration check

	    // Get size of the array.
	    #si_OutfeedsNumber := "FC_GetNrOfArrayEl"(#iqa_OutfeedsStatus);

	    // Check configuration
	    #sx_ConfigurationError := (#i_UDT_DiverterArmConfig.VerticalConveyorMode <= 0)
	    OR (#i_UDT_DiverterArmConfig.VerticalConveyorMode > 2)
	    OR (#i_UDT_DiverterArmConfig.ArmDiverterSpeedSetpointLow <= 0)
	    OR (#i_UDT_DiverterArmConfig.ArmDiverterSpeedSetpointNominal <= 0)
	    OR (#i_UDT_DiverterArmConfig.DecisionPoint <= 0)
	    OR (#i_UDT_DiverterArmConfig.ParcelFreeWindowStart <= 0)
	    OR (#i_UDT_DiverterArmConfig.ParcelFreeWindowEnd <= 0)
	    OR (#i_UDT_DiverterArmConfig.DataTransferPoint <= 0)
	    OR (#i_UDT_DiverterArmConfig.MaximumMovementTime <= 0)
	    OR (#i_UDT_DiverterArmConfig.DischargeLocationID < #ci_DestinationNumberMin)
	    OR (#i_UDT_DiverterArmConfig.DischargeLocationID > #ci_DestinationNumberMax)
	    OR (#i_UDT_DiverterArmConfig.OutfeedsNumber <= 0)
	    OR (#i_UDT_DiverterArmConfig.OutfeedsNumber > #ci_OutfeedNumberMax)
	    OR (#si_OutfeedsNumber > #ci_OutfeedNumberMax);

	END_REGION

	REGION 3 - Parcel location

	    //Save GIN number
	    IF #si_LocationGIN <> #iqa_AssociatedTrackingData[#i_UDT_DiverterArmConfig.DecisionPoint]
	        AND NOT (#iqa_AssociatedTrackingData[#i_UDT_DiverterArmConfig.DecisionPoint] = 0)
	    THEN

	        #si_LocationGIN := #iqa_AssociatedTrackingData[#i_UDT_DiverterArmConfig.DecisionPoint];

	    END_IF;

	    IF #iqa_AssociatedTrackingData[#i_UDT_DiverterArmConfig.DecisionPoint] <> 0 THEN
	        //Copy current parcel location to DB_GIN
	        "DB_GIN".GIN[#iqa_AssociatedTrackingData[#i_UDT_DiverterArmConfig.DecisionPoint]].DHL.ParcelLocation.Current := #i_UDT_DiverterArmConfig.DischargeLocationID;
	    END_IF;

	    //Check when the package leaving the "decision point"
	    #R_TRIG_ParcelLocation(CLK := #iqa_AssociatedTrackingData[#i_UDT_DiverterArmConfig.DecisionPoint] = 0);

	    IF #R_TRIG_ParcelLocation.Q AND #si_LocationGIN > 0 THEN

	        //Reset value
	        "DB_GIN".GIN[#si_LocationGIN].DHL.ParcelLocation.Current := 0;
	        //Save last position
	        "DB_GIN".GIN[#si_LocationGIN].DHL.ParcelLocation.Last := #i_UDT_DiverterArmConfig.DischargeLocationID;

	    END_IF;

	END_REGION

	REGION 2 - Decision Point

	    IF NOT #sx_ConfigurationError
	        AND NOT #sx_Disabled
	        AND #iqa_AssociatedTrackingData[#i_UDT_DiverterArmConfig.DecisionPoint] > 0
	    THEN


	        IF #si_DecisionPointGIN <> #iqa_AssociatedTrackingData[#i_UDT_DiverterArmConfig.DecisionPoint] THEN
	            #si_DecisionPointGIN := #iqa_AssociatedTrackingData[#i_UDT_DiverterArmConfig.DecisionPoint];
	            //Reset
	            #si_DecisionPointGINDistance := 0;
	        ELSIF #si_DecisionPointGIN = #iqa_AssociatedTrackingData[#i_UDT_DiverterArmConfig.DecisionPoint] THEN
	            //Count up distance
	            #si_DecisionPointGINDistance += #iq_UDT_AssociatedConveyorInterface.Displacement;
	        END_IF;


	        //New parcel
	        IF ("DB_GIN".GIN[#iqa_AssociatedTrackingData[#i_UDT_DiverterArmConfig.DecisionPoint]].DHL.ObjectID <> #ss_SortedObjectID)
	            AND #si_DecisionPointGINDistance < #i_UDT_DiverterArmConfig.DecisionParcelWindow
	            AND #sx_ActualArmPositionHome
	        THEN

	            //Check the area where the arm moves to ensure there isn't a package there
	            FOR #ti_LoopParcelFreeArea := #i_UDT_DiverterArmConfig.ParcelFreeWindowStart TO #i_UDT_DiverterArmConfig.ParcelFreeWindowEnd DO

	                //Area occupied by another parcel
	                IF #iqa_AssociatedTrackingData[#ti_LoopParcelFreeArea] > 0
	                    AND NOT (#iqa_AssociatedTrackingData[#ti_LoopParcelFreeArea] = #iqa_AssociatedTrackingData[#i_UDT_DiverterArmConfig.DecisionPoint])
	                THEN

	                    //Another parcel is within the range of arm movement. The parcel cannot be sorted.
	                    #sx_ParcelInWindow := TRUE;

	                    //Counter only for statistics
	                    #ss_Counter.ParcelDetected += 1;

	                END_IF;

	            END_FOR;

	            //Check window after sort parcel
	            IF #i_UDT_DiverterArmConfig.ParcelFreeWindow > 0 THEN

	                //Find end of parcel in tracking
	                FOR #ti_LoopParcelFreeArea := 0 TO DINT_TO_INT(#i_UDT_DiverterArmConfig.AssociatedConveyorLength) DO

	                    IF #iqa_AssociatedTrackingData[#ti_LoopParcelFreeArea] = #iqa_AssociatedTrackingData[#i_UDT_DiverterArmConfig.DecisionPoint]
	                        AND #si_SortParcelEndPositon < #ti_LoopParcelFreeArea
	                    THEN

	                        #si_SortParcelEndPositon := #ti_LoopParcelFreeArea;

	                    END_IF;

	                END_FOR;

	                //Check if from sort parcel to the next parcel is enough place
	                FOR #ti_LoopParcel := #si_SortParcelEndPositon TO #si_SortParcelEndPositon + #i_UDT_DiverterArmConfig.ParcelFreeWindow DO

	                    IF #iqa_AssociatedTrackingData[#ti_LoopParcel] <> 0
	                        AND NOT (#iqa_AssociatedTrackingData[#ti_LoopParcel] = #iqa_AssociatedTrackingData[#i_UDT_DiverterArmConfig.DecisionPoint])
	                    THEN

	                        //Another parcel is within the range of arm movement. The parcel cannot be sorted.
	                        #sx_ParcelInWindow := TRUE;

	                        //Counter only for statistics
	                        #ss_Counter.ParcelDetected += 1;

	                    END_IF;

	                END_FOR;

	                //Reset
	                #si_SortParcelEndPositon := 0;

	            END_IF;

	            IF NOT #sx_ParcelInWindow THEN

	                //A new parcel is found check the destination
	                #sx_NewParcel := True;
	                //Copy Object ID to static memory
	                #ss_SortedObjectID := "DB_GIN".GIN[#iqa_AssociatedTrackingData[#i_UDT_DiverterArmConfig.DecisionPoint]].DHL.ObjectID;
	                #si_GINSort := #iqa_AssociatedTrackingData[#i_UDT_DiverterArmConfig.DecisionPoint];
	                //Counter only for statistics
	                #ss_Counter.ParcelDetected += 1;

	            END_IF;

	            // Reset
	            #sx_ParcelInWindow := False;

	        END_IF;

	        REGION 2.1 - Sort Strategy - Sequence - Highest priority available
	            //Add sort strategy - highest priority
	            //
	            //Add generation points

	            IF "DB_GIN".GIN[#si_GINSort].DHL.SortStrategy = #cs_SortStrategyHighestPriority AND #sx_NewParcel THEN

	                //Check if the destination matches the parcel.
	                FOR #ti_LoopDestination := 1 TO 6 DO

	                    IF "DB_GIN".GIN[#si_GINSort].DHL.Destination[#ti_LoopDestination].ID = #i_UDT_DiverterArmConfig.DischargeLocationID THEN

	                        //The point is on the list of destinations
	                        #sx_GenerationMessage := TRUE;

	                    END_IF;

	                END_FOR;

	                IF #sx_GenerationMessage THEN

	                    //A loop to search the destination structure for the parcel.
	                    FOR #ti_LoopDestination := 1 TO 6 DO

	                        //A loop to search the Outfeeds status structure
	                        FOR #ti_LoopOutfeeds := 1 TO 5 DO

	                            //Check destination
	                            IF ("DB_GIN".GIN[#si_GINSort].DHL.Destination[#ti_LoopDestination].ID = #iqa_OutfeedsStatus[#ti_LoopOutfeeds].ID)
	                            THEN

	                                IF ("DB_GIN".GIN[#si_GINSort].DHL.Destination[#ti_LoopDestination].ID = #i_UDT_DiverterArmConfig.DischargeLocationID)
	                                THEN

	                                    //Check if the package can be sorted
	                                    IF (NOT #iqa_OutfeedsStatus[#ti_LoopOutfeeds].NotAvailable)
	                                        AND (NOT #iqa_OutfeedsStatus[#ti_LoopOutfeeds].Full)
	                                        AND (NOT #iqa_OutfeedsStatus[#ti_LoopOutfeeds].Disable)
	                                    THEN

	                                        //Variable trigger - this parcel should be sorted.
	                                        #sx_AutoArmDivert := TRUE;
	                                        #sx_AutoArmHome := FALSE;

	                                        //Set
	                                        "DB_GIN".GIN[#si_GINSort].DHL.Destination[#ti_LoopDestination].SortCommandActive := True;

	                                        //Counter only for statistics
	                                        #ss_Counter.SortParcelCommand += 1;

	                                        //Exit loop
	                                        EXIT;

	                                        //Generation a message why the parcel has not been sorted
	                                    ELSIF (#iqa_OutfeedsStatus[#ti_LoopOutfeeds].NotAvailable)
	                                        OR (#iqa_OutfeedsStatus[#ti_LoopOutfeeds].Full)
	                                        OR (#iqa_OutfeedsStatus[#ti_LoopOutfeeds].Disable)
	                                    THEN

	                                        //Generate a message to MFC why the parcel has not been sorted
	                                        IF #iqa_OutfeedsStatus[#ti_LoopOutfeeds].NotAvailable
	                                            OR #iqa_OutfeedsStatus[#ti_LoopOutfeeds].Disable
	                                        THEN

	                                            #FB_MFC_Sort_SortResult(is_ObjectID := "DB_GIN".GIN[#si_GINSort].DHL.ObjectID,
	                                                                    ii_DischargeLocation := #iqa_OutfeedsStatus[#ti_LoopOutfeeds].ID,
	                                                                    ii_Result := 2,
	                                                                    ii_Reason := 3,
	                                                                    ii_SourceNode := #ii_SourceNode,
	                                                                    ii_DestinationNode := #ii_DestinationNode,
	                                                                    iq_UDT_FifoHeader := #iq_UDT_FifoHeader_MFCMessage,
	                                                                    iqs_FifoData := #iqs_FifoData_MFCMessage,
	                                                                    iqdi_MessageSequenceNumber := #iqdi_MessageSequenceNumber);

	                                            //Save data in DB_GIN
	                                            "DB_GIN".GIN[#si_GINSort].DHL.Destination[#ti_LoopDestination].Rejected := True;
	                                            "DB_GIN".GIN[#si_GINSort].DHL.Destination[#ti_LoopDestination].Reason := 3;

	                                            //Counter only for statistics
	                                            #ss_Counter.SortResultMessage += 1;

	                                        END_IF;

	                                        //Generate a message to MFC why the parcel has not been sorted
	                                        IF #iqa_OutfeedsStatus[#ti_LoopOutfeeds].Full THEN

	                                            #FB_MFC_Sort_SortResult(is_ObjectID := "DB_GIN".GIN[#si_GINSort].DHL.ObjectID,
	                                                                    ii_DischargeLocation := #iqa_OutfeedsStatus[#ti_LoopOutfeeds].ID,
	                                                                    ii_Result := 2,
	                                                                    ii_Reason := 2,
	                                                                    ii_SourceNode := #ii_SourceNode,
	                                                                    ii_DestinationNode := #ii_DestinationNode,
	                                                                    iq_UDT_FifoHeader := #iq_UDT_FifoHeader_MFCMessage,
	                                                                    iqs_FifoData := #iqs_FifoData_MFCMessage,
	                                                                    iqdi_MessageSequenceNumber := #iqdi_MessageSequenceNumber);

	                                            //Save data in DB_GIN
	                                            "DB_GIN".GIN[#si_GINSort].DHL.Destination[#ti_LoopDestination].Rejected := True;
	                                            "DB_GIN".GIN[#si_GINSort].DHL.Destination[#ti_LoopDestination].Reason := 2;

	                                            //Counter only for statistics
	                                            #ss_Counter.SortResultMessage += 1;

	                                        END_IF;


	                                    END_IF;

	                                    //Generation a message why the parcel has not been sorted
	                                ELSIF (#iqa_OutfeedsStatus[#ti_LoopOutfeeds].NotAvailable)
	                                    OR (#iqa_OutfeedsStatus[#ti_LoopOutfeeds].Full)
	                                    OR (#iqa_OutfeedsStatus[#ti_LoopOutfeeds].Disable)
	                                THEN

	                                    //Generate a message to MFC why the parcel has not been sorted
	                                    IF #iqa_OutfeedsStatus[#ti_LoopOutfeeds].NotAvailable
	                                        OR #iqa_OutfeedsStatus[#ti_LoopOutfeeds].Disable
	                                    THEN

	                                        #FB_MFC_Sort_SortResult(is_ObjectID := "DB_GIN".GIN[#si_GINSort].DHL.ObjectID,
	                                                                ii_DischargeLocation := #iqa_OutfeedsStatus[#ti_LoopOutfeeds].ID,
	                                                                ii_Result := 2,
	                                                                ii_Reason := 3,
	                                                                ii_SourceNode := #ii_SourceNode,
	                                                                ii_DestinationNode := #ii_DestinationNode,
	                                                                iq_UDT_FifoHeader := #iq_UDT_FifoHeader_MFCMessage,
	                                                                iqs_FifoData := #iqs_FifoData_MFCMessage,
	                                                                iqdi_MessageSequenceNumber := #iqdi_MessageSequenceNumber);


	                                        //Save data in DB_GIN
	                                        "DB_GIN".GIN[#si_GINSort].DHL.Destination[#ti_LoopDestination].Rejected := True;
	                                        "DB_GIN".GIN[#si_GINSort].DHL.Destination[#ti_LoopDestination].Reason := 3;

	                                        //Counter only for statistics
	                                        #ss_Counter.SortResultMessage += 1;

	                                    END_IF;

	                                    //Generate a message to MFC why the parcel has not been sorted
	                                    IF #iqa_OutfeedsStatus[#ti_LoopOutfeeds].Full THEN

	                                        #FB_MFC_Sort_SortResult(is_ObjectID := "DB_GIN".GIN[#si_GINSort].DHL.ObjectID,
	                                                                ii_DischargeLocation := #iqa_OutfeedsStatus[#ti_LoopOutfeeds].ID,
	                                                                ii_Result := 2,
	                                                                ii_Reason := 2,
	                                                                ii_SourceNode := #ii_SourceNode,
	                                                                ii_DestinationNode := #ii_DestinationNode,
	                                                                iq_UDT_FifoHeader := #iq_UDT_FifoHeader_MFCMessage,
	                                                                iqs_FifoData := #iqs_FifoData_MFCMessage,
	                                                                iqdi_MessageSequenceNumber := #iqdi_MessageSequenceNumber);


	                                        //Save data in DB_GIN
	                                        "DB_GIN".GIN[#si_GINSort].DHL.Destination[#ti_LoopDestination].Rejected := True;
	                                        "DB_GIN".GIN[#si_GINSort].DHL.Destination[#ti_LoopDestination].Reason := 2;

	                                        //Counter only for statistics
	                                        #ss_Counter.SortResultMessage += 1;

	                                    END_IF;


	                                    // Check if the 'HigherPriority' destination is available
	                                ELSIF (NOT #iqa_OutfeedsStatus[#ti_LoopOutfeeds].NotAvailable)
	                                    AND (NOT #iqa_OutfeedsStatus[#ti_LoopOutfeeds].Full)
	                                    AND (NOT #iqa_OutfeedsStatus[#ti_LoopOutfeeds].Disable)
	                                    AND ("DB_GIN".GIN[#si_GINSort].DHL.Destination[#ti_LoopDestination].ID < #i_UDT_DiverterArmConfig.DischargeLocationID)
	                                THEN

	                                    //Set variable 'HigherPriorityAvailable'
	                                    #ss_SortStrategy.HigherPriorityAvailable := TRUE;
	                                    #ss_SortStrategy.ObjectID := "DB_GIN".GIN[#si_GINSort].DHL.ObjectID;

	                                    //Exit loop
	                                    EXIT;

	                                END_IF;

	                            END_IF;

	                        END_FOR;

	                        //Check if the package can be sorted or higher piority destination available
	                        //Release the loop
	                        IF #sx_AutoArmDivert
	                            OR #ss_SortStrategy.HigherPriorityAvailable
	                        THEN

	                            //Counter only for statistics
	                            #ss_Counter.LoopExit += 1;

	                            EXIT;

	                        END_IF;

	                    END_FOR;

	                    //  Generation message - Higher priority available
	                    IF #ss_SortStrategy.HigherPriorityAvailable THEN

	                        #FB_MFC_Sort_SortResult_HigherPriorityAvailable(is_ObjectID := #ss_SortStrategy.ObjectID,
	                                                                        ii_DischargeLocation := #i_UDT_DiverterArmConfig.DischargeLocationID,
	                                                                        ii_Result := 2,
	                                                                        ii_Reason := 7,
	                                                                        ii_SourceNode := #ii_SourceNode,
	                                                                        ii_DestinationNode := #ii_DestinationNode,
	                                                                        iq_UDT_FifoHeader := #iq_UDT_FifoHeader_MFCMessage,
	                                                                        iqs_FifoData := #iqs_FifoData_MFCMessage,
	                                                                        iqdi_MessageSequenceNumber := #iqdi_MessageSequenceNumber);


	                        //Save data in DB_GIN
	                        "DB_GIN".GIN[#si_GINSort].DHL.Destination[#ti_LoopDestination].Rejected := True;
	                        "DB_GIN".GIN[#si_GINSort].DHL.Destination[#ti_LoopDestination].Reason := 7;

	                        //Reset
	                        #ss_SortStrategy.HigherPriorityAvailable := False;
	                        #ss_SortStrategy.ObjectID := '';

	                        //Counter only for statistics
	                        #ss_Counter.SortResultMessage += 1;

	                    END_IF;

	                END_IF;

	                //Reset
	                #sx_GenerationMessage := False;

	                //Reset value
	                #sx_NewParcel := False;

	            END_IF;

	        END_REGION

	        REGION 2.2 - Sort Strategy - OrderOfProximity - Nearest

	            IF "DB_GIN".GIN[#si_GINSort].DHL.SortStrategy = #cs_SortStrategyNearest AND #sx_NewParcel THEN

	                //Destination
	                FOR #ti_LoopDestinationNearest := 0 TO #ci_OutfeedNumberMax DO

	                    IF "DB_GIN".GIN[#si_GINSort].General.Destination[#ti_LoopDestinationNearest] = #i_UDT_DiverterArmConfig.DischargeLocationID
	                        AND NOT #iqa_OutfeedsStatus[#i_UDT_DiverterArmConfig.OutfeedsNumber].NotAvailable
	                        AND NOT #iqa_OutfeedsStatus[#i_UDT_DiverterArmConfig.OutfeedsNumber].Full
	                        AND NOT #iqa_OutfeedsStatus[#i_UDT_DiverterArmConfig.OutfeedsNumber].Disable
	                        AND #iq_UDT_ExitConveyorHandshake.RTR

	                    THEN

	                        //Variable trigger - this parcel should be sorted.
	                        #sx_AutoArmDivert := TRUE;
	                        #sx_AutoArmHome := FALSE;


	                        //Message to MFC generation and copy data to DB_GIN

	                        //Exit the loop
	                        EXIT;

	                    END_IF;

	                END_FOR;

	                //Reset value
	                #sx_NewParcel := False;

	            END_IF;

	        END_REGION

	    END_IF;

	END_REGION

	REGION 3 - Diverter arm handling

	    REGION 3.1 - Movement conditions

	        //Conditions to set bit sx_Ready to operate in automatic mode
	        #sx_Ready := #ix_SafetyOk                                               // Safety signalling
	        AND #ix_24vOk                                                           // 24V
	        AND #ix_400vOk                                                          // 400V
	        AND #ix_HardwareOk                                                      // PNPN device
	        AND NOT #iq_UDT_ArmConveyorInterface.ConfigurationError;                // No configuration error

	        //Share HardwareOK signal over interface
	        #iq_UDT_ArmConveyorInterface.HardwareOk := #ix_HardwareOk;

	        ///Conditions from other items
	        #sx_SwitchEnable := NOT #s_UDT_CommonStatus.Error;                       // Error present

	        //Command to stop Associated conveyor
	        #qx_AssociatedConveyorHold := (#iq_UDT_VerticalConveyorInterface.InternalErrorVFD AND NOT #sx_ActualArmPositionHome)              // Vertical conveyor
	        OR (#sx_ActualArmPositionDivert AND (NOT #iq_UDT_ExitConveyorHandshake.RTR));                                                     // Exit conveyor redy to receive parcels

	    END_REGION

	    REGION 3.2 -Sensor

	        //Sensors reached
	        // Limit switch home position
	        //Set
	        IF NOT #sx_LS_HomeFiltered AND #iq_UDT_ArmConveyorInterface.RunFwd THEN
	            #sx_LimitSwitchHomeReached := True;
	        END_IF;
	        //Reset
	        IF (#iq_UDT_ArmConveyorInterface.RunRvs AND #R_TRIG_LS_Home.Q)
	            OR (NOT #iq_UDT_ArmConveyorInterface.VFDRunning AND #R_TRIG_LS_Home.Q)
	        THEN
	            #sx_LimitSwitchHomeReached := False;
	        END_IF;

	        //Limit switch divert position
	        IF NOT #sx_LS_DivertFiltered AND #iq_UDT_ArmConveyorInterface.RunRvs THEN
	            #sx_LimitSwitchDivertReached := True;
	        END_IF;
	        //Reset
	        IF (#iq_UDT_ArmConveyorInterface.RunFwd AND #R_TRIG_LS_Divert.Q)
	            OR (NOT #iq_UDT_ArmConveyorInterface.VFDRunning AND #R_TRIG_LS_Divert.Q)
	        THEN
	            #sx_LimitSwitchDivertReached := False;
	        END_IF;

	        // Home position
	        //Set
	        IF NOT #sx_PRX_HomeFiltered AND #iq_UDT_ArmConveyorInterface.RunFwd THEN
	            #sx_PositionHomeReached := True;
	        END_IF;
	        //Reset
	        IF (#iq_UDT_ArmConveyorInterface.RunRvs AND #R_TRIG_PRX_Home.Q)
	            OR (NOT #iq_UDT_ArmConveyorInterface.VFDRunning AND #R_TRIG_PRX_Home.Q)
	        THEN
	            #sx_PositionHomeReached := False;
	        END_IF;

	        //Divert position
	        IF NOT #sx_PRX_DivertFiltered AND #iq_UDT_ArmConveyorInterface.RunRvs THEN
	            #sx_PositionDivertReached := True;
	        END_IF;
	        //Reset
	        IF (#iq_UDT_ArmConveyorInterface.RunFwd AND #R_TRIG_PRX_Divert.Q)
	            OR (NOT #iq_UDT_ArmConveyorInterface.VFDRunning AND #R_TRIG_PRX_Divert.Q)
	        THEN
	            #sx_PositionDivertReached := False;
	        END_IF;

	    END_REGION

	    REGION 3.3 - Automatic movement conditions

	        //Home position
	        #sx_MoveToHomePosition := #sx_Ready                  //Conditions for movement
	        AND #sx_SwitchEnable                                 //
	        AND #iq_UDT_EquipmentControl.Command.AutomaticOn     //
	        AND NOT #iq_UDT_ArmDiverterCommand.ManualMode        //
	        AND #sx_PRX_HomeFiltered                             //
	        AND NOT #sx_PositionHomeReached                      //
	        AND #sx_AutoArmHome                                  //Arm return signal to Home position
	        AND NOT #sx_AutoArmDivert                            //
	        AND (NOT #iq_UDT_EquipmentControl.Command.StopRequest OR #sx_MoveToHomePosition);

	        //Divert position
	        #sx_MoveToDivertPosition := #sx_Ready                //Conditions for movement
	        AND #sx_SwitchEnable                                 //
	        AND #iq_UDT_EquipmentControl.Command.AutomaticOn     //
	        AND NOT #iq_UDT_ArmDiverterCommand.ManualMode        //
	        AND #sx_PRX_DivertFiltered                           //
	        AND NOT #sx_PositionDivertReached                    //
	        AND NOT #sx_AutoArmHome                              //
	        AND #sx_AutoArmDivert                                //Sort conditions active
	        AND (NOT #iq_UDT_EquipmentControl.Command.StopRequest OR #sx_MoveToDivertPosition);

	        //Reset automatic control command when manual mode
	        IF #iq_UDT_ArmDiverterCommand.ManualMode THEN
	            #sx_AutoArmHome := False;
	            #sx_AutoArmDivert := False;
	        END_IF;

	    END_REGION

	    REGION 3.4 - Manual mode

	        //Home position
	        IF
	            #sx_PRX_HomeFiltered                                   //The position sensor doesn't detect the arm
	            AND #iq_UDT_ArmDiverterCommand.ManualMode              //Manual mode active
	            AND #iq_UDT_ArmDiverterCommand.ManualHomePosition      //Go to home position active
	        THEN
	            #sx_ManualToHomePosition := TRUE;
	        END_IF;

	        //Reset
	        IF (NOT #iq_UDT_ArmDiverterCommand.ManualMode)
	            OR #s_UDT_CommonStatus.Error
	            OR (NOT #sx_PRX_HomeFiltered)
	            OR #sx_LimitSwitchHomeReached
	            OR #sx_PositionHomeReached
	        THEN
	            #sx_ManualToHomePosition := FALSE;
	        END_IF;

	        //Divert direction
	        IF #sx_PRX_DivertFiltered                                      //The position sensor doesn't detect the arm
	            AND #iq_UDT_ArmDiverterCommand.ManualMode                  //Manual mode active
	            AND #iq_UDT_ArmDiverterCommand.ManualDivertPosition        //Go to divert position active
	        THEN
	            #sx_ManualToDivertPosition := TRUE;
	        END_IF;

	        //Reset
	        IF (NOT #iq_UDT_ArmDiverterCommand.ManualMode)
	            OR #s_UDT_CommonStatus.Error
	            OR (NOT #sx_PRX_DivertFiltered)
	            OR #sx_LimitSwitchDivertReached
	            OR #sx_PositionDivertReached
	        THEN
	            #sx_ManualToDivertPosition := FALSE;
	        END_IF;

	    END_REGION

	    REGION 3.5 - Jog Mode

	        //Home direction
	        #sx_JogToHomePosition :=
	        #sx_LS_HomeFiltered                                         //The limit switch doesn't detect the arm
	        AND #sx_PRX_HomeFiltered
	        AND NOT #sx_LimitSwitchHomeReached
	        AND NOT #sx_PositionHomeReached
	        AND #iq_UDT_ArmDiverterCommand.ManualMode                   //Manual mode active
	        AND #iq_UDT_ArmDiverterCommand.JogHomePosition              //Jog to home position active
	        AND NOT #iq_UDT_ArmDiverterCommand.JogDivertPosition;       //

	        //Divert direction
	        #sx_JogToDivertPosition :=
	        #sx_LS_DivertFiltered                                      //The limit switch doesn't detect the arm
	        AND #sx_PRX_DivertFiltered
	        AND NOT #sx_LimitSwitchDivertReached
	        AND NOT #sx_PositionDivertReached
	        AND #iq_UDT_ArmDiverterCommand.ManualMode                  //Manual mode active
	        AND #iq_UDT_ArmDiverterCommand.JogDivertPosition           //Jog to divert position active
	        AND (NOT #iq_UDT_ArmDiverterCommand.JogHomePosition);

	        // Detecting rising edge on manual jog Home
	        #R_TRIG_ManualJogHome(CLK := #sx_JogToHomePosition);

	        // Detecting rising edge on manual jog Divert
	        #R_TRIG_ManualJogDivert(CLK := #sx_JogToDivertPosition);

	        IF #iq_UDT_ArmDiverterCommand.ManualMode                                        // Conditions to run in manual mode
	            AND (#R_TRIG_ManualJogHome.Q                                                  // Trigger to start VSU run in manual jog mode UP
	            OR #R_TRIG_ManualJogDivert.Q)                                                 // Trigger to start VSU run in manual jog mode Down
	            AND NOT #s_FB_Jog_Enable.qx_DelayedSignal
	        THEN

	            #iq_UDT_EquipmentControl.Request.SignalingRequest := TRUE;                  // Request signaling TO control block before VSU runs in manual mode

	        END_IF;

	        // Time to start without start warning while jogging
	        #s_FB_Jog_Enable(iudi_OffDelayTime := #i_UDT_DiverterArmConfig.JogNoHornTime,
	                         ix_SignalToDelay := #sx_JogToDivertPosition OR #sx_JogToHomePosition);

	    END_REGION

	    REGION 3.6 - Arm conveyor - Low speed

	        //Set
	        IF (#sx_MoveToHomePosition AND #R_TRIG_BRK_PRX_Home.Q)
	            OR (#sx_MoveToDivertPosition AND #R_TRIG_BRK_PRX_Divert.Q)
	            OR (#sx_ManualToHomePosition AND #R_TRIG_BRK_PRX_Home.Q)
	            OR (#sx_ManualToDivertPosition AND #R_TRIG_BRK_PRX_Divert.Q)
	        THEN
	            #sx_ArmDiverterLowSpeed := TRUE;
	        END_IF;

	        //Trigger
	        #F_TRIG_ArmConveyorLowSpeed(CLK := #sx_MoveToHomePosition OR #sx_MoveToDivertPosition OR #sx_ManualToHomePosition OR #sx_ManualToDivertPosition);

	        //Reset
	        IF #F_TRIG_ArmConveyorLowSpeed.Q
	        THEN
	            #sx_ArmDiverterLowSpeed := FALSE;
	        END_IF;

	    END_REGION

	    REGION 3.7 - Copy command to VFD Interface

	        //Vertical speed handling
	        IF #sx_ArmDiverterLowSpeed OR #sx_JogToHomePosition OR #sx_JogToDivertPosition THEN
	            #iq_UDT_ArmConveyorInterface.SpeedSetpoint := #i_UDT_DiverterArmConfig.ArmDiverterSpeedSetpointLow;
	        ELSE
	            #iq_UDT_ArmConveyorInterface.SpeedSetpoint := #i_UDT_DiverterArmConfig.ArmDiverterSpeedSetpointNominal;
	        END_IF;

	        //Directions
	        #iq_UDT_ArmConveyorInterface.RunFwd := #sx_MoveToHomePosition       //Automatic mode
	        OR #sx_ManualToHomePosition                                         //Manual mode
	        OR #sx_JogToHomePosition;                                           //Jog mode

	        #iq_UDT_ArmConveyorInterface.RunRvs := #sx_MoveToDivertPosition     //Automatic mode
	        OR #sx_ManualToDivertPosition                                       //Manual mode
	        OR #sx_JogToDivertPosition;                                         //Jog mode

	    END_REGION

	    REGION 3.8 - Return conditions

	        IF #sx_ActualArmPositionDivert THEN
	            #sx_AutoArmDivert := FALSE;
	        END_IF;

	        //Check that the package has been sorted correctly
	        IF #sx_ActualArmPositionDivert
	        THEN

	            //Return conditions
	            IF #R_TRIG_ExitSensor.Q
	            THEN

	                #sx_AutoArmHome := TRUE;

	                //Save information in "DB_GIN"
	                FOR #ti_LoopResult := 1 TO 6 DO

	                    IF "DB_GIN".GIN[#si_GINSort].DHL.Destination[#ti_LoopResult].ID = #i_UDT_DiverterArmConfig.DischargeLocationID THEN
	                        "DB_GIN".GIN[#si_GINSort].DHL.Destination[#ti_LoopResult].ParcelSorted := True;
	                    END_IF;

	                END_FOR;

	                ///Generation message to MFC
	                #FB_MFC_Sort_SortResult(is_ObjectID := #ss_SortedObjectID,
	                                        ii_DischargeLocation := #i_UDT_DiverterArmConfig.DischargeLocationID,
	                                        ii_Result := 1,
	                                        ii_Reason := 1,
	                                        ii_SourceNode := #ii_SourceNode,
	                                        ii_DestinationNode := #ii_DestinationNode,
	                                        iq_UDT_FifoHeader := #iq_UDT_FifoHeader_MFCMessage,
	                                        iqs_FifoData := #iqs_FifoData_MFCMessage,
	                                        iqdi_MessageSequenceNumber := #iqdi_MessageSequenceNumber);

	            END_IF;

	            // Reset value
	            #sx_ParcelSorted := False;

	        END_IF;

	        //Reset variable return when arm is at home position
	        IF NOT #sx_PRX_HomeFiltered THEN
	            #sx_AutoArmHome := FALSE;
	        END_IF;

	    END_REGION

	    REGION 3.9 - Arm movement check, positons check

	        //Position Home
	        #sx_ActualArmPositionHome := (NOT #sx_PRX_HomeFiltered) AND #ix_HardwareOk;

	        //On way
	        #sx_ActualArmPositionOnWay := #sx_LS_HomeFiltered AND #sx_LS_DivertFiltered AND #sx_PRX_HomeFiltered AND #sx_PRX_DivertFiltered AND #iq_UDT_ArmConveyorInterface.VFDRunning;

	        //Position Divert
	        #sx_ActualArmPositionDivert := (NOT #sx_PRX_DivertFiltered) AND #ix_HardwareOk;

	    END_REGION

	    REGION 3.10 - Vertical conveyor

	        CASE #i_UDT_DiverterArmConfig.VerticalConveyorMode OF

	            1:  //[1]Continuous operation if the main conveyor is running
	                #qx_VerticalConveyorHold := NOT #iq_UDT_AssociatedConveyorInterface.VFDRunning;

	            2:  //[2]Operation if the main conveyor is running and  arm is not in Home position
	                #qx_VerticalConveyorHold := NOT #iq_UDT_AssociatedConveyorInterface.VFDRunning
	                OR NOT #sx_PRX_HomeFiltered;

	        END_CASE;

	    END_REGION

	    REGION 3.11 - Errors & inhibit stop

	        // Reset signal is sent to the interface Arm (VFD block)
	        #iq_UDT_ArmConveyorInterface.InternalErrorReset := #iq_UDT_EquipmentControl.Command.Reset;
	        #iq_UDT_ArmConveyorInterface.ResetStatistics := #iq_UDT_EquipmentControl.Command.ResetData;

	        //Error
	        #s_UDT_CommonStatus.Error := #iq_UDT_ArmConveyorInterface.InternalErrorVFD               // Internal VFD error status
	        OR #iq_UDT_ArmConveyorInterface.Disconnected                                            // Isolator switch error status
	        OR #s_UDT_HMIStatus.Specific.LimitDivertError
	        OR #s_UDT_HMIStatus.Specific.LimitHomeError
	        OR #s_UDT_HMIStatus.Specific.PXDivertError
	        OR #s_UDT_HMIStatus.Specific.PXHomeError
	        OR #s_UDT_HMIStatus.Specific.ReferencError
	        OR #s_UDT_HMIStatus.Specific.TimeoutError;

	        //Warning
	        #s_UDT_CommonStatus.Warning := #iq_UDT_ArmConveyorInterface.InternalWarningVFD;        //Internal Warning VFD added

	        //Movement timeout error
	        #s_FB_TimeoutError(iudi_OnDelayTime := #i_UDT_DiverterArmConfig.MaximumMovementTime,
	                           ix_SignalToDelay := ((#sx_MoveToHomePosition AND #sx_PRX_HomeFiltered) OR (#sx_MoveToDivertPosition AND #sx_PRX_DivertFiltered)));

	        IF #s_FB_TimeoutError.qx_DelayedSignal THEN
	            #s_UDT_HMIStatus.Specific.TimeoutError := True;
	        END_IF;

	        //Reference error - The arm does not move and any of the sensors detect it
	        IF NOT #iq_UDT_ArmConveyorInterface.VFDRunning
	            AND #sx_LS_HomeFiltered
	            AND #sx_LS_DivertFiltered
	            AND #sx_PRX_HomeFiltered
	            AND #sx_PRX_DivertFiltered
	        THEN
	            #s_UDT_HMIStatus.Specific.ReferencError := True;
	        END_IF;

	        //Sensor errors
	        //Movement command active
	        #s_FB_InhibitTimeFilter(iudi_OffDelayTime := #cudi_InhibitTimeFilterTimeOFF,
	                                ix_SignalToDelay := (#iq_UDT_ArmConveyorInterface.RunRvs
	                                OR #iq_UDT_ArmConveyorInterface.RunFwd
	                                OR #iq_UDT_ArmConveyorInterface.ActualSpeed <> 0),
	                                ix_Enable := TRUE,
	                                qx_DelayedSignal => #tx_MovementCommandActive);

	        // #tx_MovementCommandActive := (#iq_UDT_ArmConveyorInterface.RunRvs
	        // OR #iq_UDT_ArmConveyorInterface.RunFwd
	        // OR #iq_UDT_ArmConveyorInterface.ActualSpeed <> 0);
	        //  //OR #s_FB_DivertTime.qx_DelayedSignal

	        //Movement command active,copy value to EquipmentControl structure
	        #iq_UDT_EquipmentControl.Request.InhibitStop := #iq_UDT_EquipmentControl.Request.InhibitStop OR #tx_MovementCommandActive;

	        // Limit swich sensor error
	        IF NOT #tx_MovementCommandActive AND (#R_TRIG_LS_Home.Q OR #F_TRIG_LS_Home.Q) THEN
	            #s_UDT_HMIStatus.Specific.LimitHomeError := True;
	        END_IF;
	        //Limit swich sensor error
	        IF NOT #tx_MovementCommandActive AND (#R_TRIG_LS_Divert.Q OR #F_TRIG_LS_Divert.Q) THEN
	            #s_UDT_HMIStatus.Specific.LimitDivertError := True;
	        END_IF;
	        //Proxy sensor error
	        IF NOT #tx_MovementCommandActive AND (#R_TRIG_LS_Home.Q OR #F_TRIG_LS_Home.Q) THEN
	            #s_UDT_HMIStatus.Specific.PXHomeError := True;
	        END_IF;
	        //Proxy sensor error
	        IF NOT #tx_MovementCommandActive AND (#R_TRIG_LS_Divert.Q OR #F_TRIG_LS_Divert.Q) THEN
	            #s_UDT_HMIStatus.Specific.PXDivertError := True;
	        END_IF;

	        //Divert Time
	        #s_FB_DivertTime(iudi_OnDelayTime := #i_UDT_DiverterArmConfig.MaximumParcelDivertTime,
	                         ix_SignalToDelay := (#sx_AutoArmDivert AND NOT #sx_ActualArmPositionHome)
	                         OR (#sx_ActualArmPositionDivert AND #iq_UDT_AssociatedConveyorInterface.VFDRunning));

	        IF #s_FB_DivertTime.qx_DelayedSignal THEN
	            #s_UDT_HMIStatus.Specific.ParcelDivertError := TRUE;
	        END_IF;

	        //Reset Errors
	        IF #iq_UDT_ArmDiverterCommand.Reset THEN
	            //Arm movement timed out
	            IF #s_UDT_HMIStatus.Specific.TimeoutError THEN
	                #s_UDT_HMIStatus.Specific.TimeoutError := FALSE;
	            END_IF;
	            //Limit swich sensor error
	            IF #s_UDT_HMIStatus.Specific.LimitHomeError THEN
	                #s_UDT_HMIStatus.Specific.LimitHomeError := FALSE;
	            END_IF;
	            //Limit swich sensor error
	            IF #s_UDT_HMIStatus.Specific.LimitDivertError THEN
	                #s_UDT_HMIStatus.Specific.LimitDivertError := FALSE;
	            END_IF;
	            //Proxy sensor error
	            IF #s_UDT_HMIStatus.Specific.PXHomeError THEN
	                #s_UDT_HMIStatus.Specific.PXHomeError := FALSE;
	            END_IF;
	            //Proxy sensor error
	            IF #s_UDT_HMIStatus.Specific.PXDivertError THEN
	                #s_UDT_HMIStatus.Specific.PXDivertError := FALSE;
	            END_IF;
	            //Referencing error
	            IF #s_UDT_HMIStatus.Specific.ReferencError
	                AND #iq_UDT_ArmDiverterCommand.ManualMode
	                AND NOT #sx_PRX_HomeFiltered
	            THEN
	                #s_UDT_HMIStatus.Specific.ReferencError := FALSE;
	            END_IF;
	            //Parcel divert error
	            IF #s_UDT_HMIStatus.Specific.ParcelDivertError THEN
	                #s_UDT_HMIStatus.Specific.ParcelDivertError := False;
	            END_IF;

	        END_IF;

	    END_REGION

	    REGION 3.12 - Status

	        //Write outfeed status
	        #iqa_OutfeedsStatus[#i_UDT_DiverterArmConfig.OutfeedsNumber].NotAvailable := (NOT #sx_Ready)
	        OR (NOT #sx_SwitchEnable); // to add more conditions

	        //Arm at home position
	        #s_UDT_HMIStatus.Specific.AtHomePosition := #sx_ActualArmPositionHome;
	        //Arm at divert position
	        #s_UDT_HMIStatus.Specific.AtDivertPosition := #sx_ActualArmPositionDivert;

	        // HMI status update
	        IF #s_UDT_CommonStatusOld <> #s_UDT_CommonStatus
	        THEN
	            // HMI status initialization
	            #s_UDT_HMIStatus.Status := 0;

	            // Energy save
	            IF #s_UDT_CommonStatus.EnergySave
	            THEN
	                #s_UDT_HMIStatus.Status := "DB_HMIStatusConfiguration".EnergySave;
	            END_IF;

	            // Running
	            IF #s_UDT_CommonStatus.Running
	            THEN
	                #s_UDT_HMIStatus.Status := "DB_HMIStatusConfiguration".Running;
	            END_IF;

	            // Stopped
	            IF #s_UDT_CommonStatus.Stopped
	            THEN
	                #s_UDT_HMIStatus.Status := "DB_HMIStatusConfiguration".Stopped;
	            END_IF;

	            // Dieback
	            IF #s_UDT_CommonStatus.Dieback
	            THEN
	                #s_UDT_HMIStatus.Status := "DB_HMIStatusConfiguration".Dieback;
	            END_IF;

	            // Halted
	            IF #s_UDT_CommonStatus.Halted
	            THEN
	                #s_UDT_HMIStatus.Status := "DB_HMIStatusConfiguration".Halted;
	            END_IF;

	            // Manual
	            IF #s_UDT_CommonStatus.Manual
	            THEN
	                #s_UDT_HMIStatus.Status := "DB_HMIStatusConfiguration".Manual;
	            END_IF;

	            // Running in manual mode
	            IF #s_UDT_CommonStatus.ManualRun
	            THEN
	                #s_UDT_HMIStatus.Status := "DB_HMIStatusConfiguration".ManualRun;
	            END_IF;

	            //Error
	            IF #s_UDT_CommonStatus.Error THEN
	                #s_UDT_HMIStatus.Status := "DB_HMIStatusConfiguration".Error;
	            END_IF;

	            // Safety stop
	            IF (#s_UDT_CommonStatus.SafetyStop)
	            THEN
	                #s_UDT_HMIStatus.Status := "DB_HMIStatusConfiguration".SafetyStop;
	            END_IF;

	            #s_UDT_CommonStatusOld := #s_UDT_CommonStatus;              // Copy status to memory
	            #q_UDT_Status := #s_UDT_CommonStatus;                       // Copy status to output

	        END_IF;

	        // Copy HMI status to output
	        #q_UDT_HMIStatus := #s_UDT_HMIStatus;

	    END_REGION

	END_REGION

	REGION 4 - Tracking data handling

	    IF #sx_ActualArmPositionDivert THEN

	        //To test on site
	        //Copy handshakes
	        //Upstream to downstream
	        #iq_UDT_ExitConveyorHandshake.GIN := #iqa_AssociatedTrackingData[#i_UDT_DiverterArmConfig.DataTransferPoint];
	        #iqa_AssociatedTrackingData[#i_UDT_DiverterArmConfig.DataTransferPoint] := 0;
	        //#iq_UDT_HandShakeConveyorExtended.NrOfPosToShift := #iq_UDT_HandShakeSorterConveyor.NrOfPosToShift;


	        #iq_UDT_ExitConveyorHandshake.RTS := #iq_UDT_AssociatedConveyorHandshake.RTS;
	        #iq_UDT_ExitConveyorHandshake.TIP := #iq_UDT_AssociatedConveyorHandshake.TIP;
	        #iq_UDT_ExitConveyorHandshake.ResetEnergySave := #iq_UDT_AssociatedConveyorHandshake.ResetEnergySave;
	        // Downstream to upstream
	        #iq_UDT_AssociatedConveyorHandshake.RTR := #iq_UDT_ExitConveyorHandshake.RTR;
	        #iq_UDT_AssociatedConveyorHandshake.DownstreamDisplacement := #iq_UDT_ExitConveyorHandshake.DownstreamDisplacement;
	        #iq_UDT_AssociatedConveyorHandshake.CascadeStartUp := #iq_UDT_ExitConveyorHandshake.CascadeStartUp;

	        // Clear GIN if there is no RTR
	        IF NOT #iq_UDT_ExitConveyorHandshake.RTR
	        THEN

	            #iq_UDT_ExitConveyorHandshake.GIN := 0;
	            #iq_UDT_ExitConveyorHandshake.NrOfPosToShift := 0;

	        END_IF;

	    END_IF;

	    //Arm diverter is not at the position, clear Handshake
	    //To test on site
	    IF NOT #sx_ActualArmPositionHome
	        AND NOT #sx_ActualArmPositionDivert
	    THEN

	        // Reset Handshake extended position downstream
	        #iq_UDT_ExitConveyorHandshake.GIN := 0;
	        #iq_UDT_ExitConveyorHandshake.NrOfPosToShift := 0;
	        #iq_UDT_ExitConveyorHandshake.RTS := FALSE;
	        #iq_UDT_ExitConveyorHandshake.TIP := FALSE;
	        #iq_UDT_ExitConveyorHandshake.DownstreamDisplacement := 0;
	        #iq_UDT_ExitConveyorHandshake.ResetEnergySave := FALSE;

	    END_IF;

	END_REGION
END_FUNCTION_BLOCK

FUNCTION_BLOCK "FB_SecurityCage"
{ S7_Optimized_Access := 'TRUE' }
VERSION : 0.1
// ATTRIBUTES
// AUTO_NUMBER = True
// BLOCK_NUMBER = 101
// END_ATTRIBUTES
   VAR_INPUT
      ix_StartStopButton { ExternalAccessible := 'False'; ExternalVisible := 'False'; ExternalWritable := 'False'} : Bool;   // Start stop push button
      ix_DirectionButton { ExternalAccessible := 'False'; ExternalVisible := 'False'; ExternalWritable := 'False'} : Bool;   // Direction push button
   END_VAR

